(* IEC 61131-3 sources: elnaProjects/ElpcLogic/PomarKc7Changed/build_USO_ecl (part 5) *)

  (* Отключение МВ1 от КНА   *)
  stSs_Ini(data_Ini := true, inverse:=TRUE, (*wait_time:=T#0S,*) str_SS := IM.SingleSignals.Nalichie_BP5);
  inits := inits + BOOL_TO_UINT(stSs_Ini.Init);

  (* Отключение МВ1 от КНА   *)
  stSs_Ini(data_Ini := true, inverse:=TRUE, (*wait_time:=T#0S,*) str_SS := IM.SingleSignals.Nalichie_BP6);
  inits := inits + BOOL_TO_UINT(stSs_Ini.Init);

  (* Отключение МВ1 от КНА   *)
  stSs_Ini(data_Ini := true, inverse:=TRUE, (*wait_time:=T#0S,*) str_SS := IM.SingleSignals.Nalichie_BP7_BP8);
  inits := inits + BOOL_TO_UINT(stSs_Ini.Init);

  (* Отключение МВ1 от КНА   *)
  stSs_Ini(data_Ini := true, inverse:=TRUE, (*wait_time:=T#0S,*) str_SS := IM.SingleSignals.Nalichie_BP9_BP10);
  inits := inits + BOOL_TO_UINT(stSs_Ini.Init);

  (* Отключение МВ1 от КНА   *)
  stSs_Ini(data_Ini := true, inverse:=TRUE, (*wait_time:=T#0S,*) str_SS := IM.SingleSignals.Nalichie_cepei_upravlen_mv);
  inits := inits + BOOL_TO_UINT(stSs_Ini.Init);

  (* Отключение МВ1 от КНА   *)
  stSs_Ini(data_Ini := true, inverse:=TRUE, (*wait_time:=T#0S,*) str_SS := IM.SingleSignals.Nalichie_220BEAO);
  inits := inits + BOOL_TO_UINT(stSs_Ini.Init);

  (* Отключение МВ1 от КНА   *)
  stSs_Ini(data_Ini := true, inverse:=TRUE, (*wait_time:=T#0S,*) str_SS := IM.SingleSignals.Nalichie_per_220_na_vhode);
  inits := inits + BOOL_TO_UINT(stSs_Ini.Init);

  (* Отключение МВ1 от КНА   *)
  stSs_Ini(data_Ini := true, inverse:=TRUE, (*wait_time:=T#0S,*) str_SS := IM.SingleSignals.Nalichie_post_220_na_vhode);
  inits := inits + BOOL_TO_UINT(stSs_Ini.Init);

  (* Отключение МВ1 от КНА   *)
  stSs_Ini(data_Ini := true, inverse:=TRUE, (*wait_time:=T#0S,*) str_SS := IM.SingleSignals.Nalichie_BP11);
  inits := inits + BOOL_TO_UINT(stSs_Ini.Init);

  (* Отключение МВ1 от КНА   *)
  stSs_Ini(data_Ini := true, inverse:=TRUE, (*wait_time:=T#0S,*) str_SS := IM.SingleSignals.Nalichie_BP12);
  inits := inits + BOOL_TO_UINT(stSs_Ini.Init);

  (* Отключение МВ1 от КНА   *)
  stSs_Ini(data_Ini := true, inverse:=TRUE, (*wait_time:=T#0S,*) str_SS := IM.SingleSignals.Dver_SHU_pered_otkrita);
  inits := inits + BOOL_TO_UINT(stSs_Ini.Init);

  (* Отключение МВ1 от КНА   *)
  stSs_Ini(data_Ini := true, inverse:=TRUE, (*wait_time:=T#0S,*) str_SS := IM.SingleSignals.Dver_SHU_zad_otkrita);
  inits := inits + BOOL_TO_UINT(stSs_Ini.Init);

  (* Отключение МВ1 от КНА   *)
  stSs_Ini(data_Ini := true, inverse:=TRUE, (*wait_time:=T#0S,*) str_SS := IM.SingleSignals.EO_GPA_ot_knopki_SHU);
  inits := inits + BOOL_TO_UINT(stSs_Ini.Init);

  (* Отключение МВ1 от КНА   *)
  stSs_Ini(data_Ini := true, inverse:=TRUE, (*wait_time:=T#0S,*) str_SS := IM.SingleSignals.EO_EGPA_ot_PRY);
  inits := inits + BOOL_TO_UINT(stSs_Ini.Init);

  (* Отключение МВ1 от КНА   *)
  stSs_Ini(data_Ini := true, inverse:=TRUE, (*wait_time:=T#0S,*) str_SS := IM.SingleSignals.Synchroniz_rezhima_K1);
  inits := inits + BOOL_TO_UINT(stSs_Ini.Init);

                                       (* Стартовая инициализация singleOutput *)
  (* Идикация НО (подсветка кнопки на шкафу)   *)
  stSo_Ini(data_Ini := true, inOpcCommandsDisabled:=TRUE, (*wait_time:=T#0S,*) str_SO := IM.SingleOutputs.Rabota_EGPA);
  inits := inits + BOOL_TO_UINT(stSo_Ini.Init);

  (* Взвод включения БЭАО по неисправности ПТС   *)
  stSo_Ini(data_Ini := true, inOpcCommandsDisabled:=TRUE, wait_time:=T#0S, str_SO := IM.SingleOutputs.Neispr_EGPA);
  inits := inits + BOOL_TO_UINT(stSo_Ini.Init);

  (* Авария ЭГПА в КЦ   *)
  stSo_Ini(data_Ini := true, inOpcCommandsDisabled:=TRUE, (*wait_time:=T#0S,*) str_SO := IM.SingleOutputs.Avary_EGPA);
  inits := inits + BOOL_TO_UINT(stSo_Ini.Init);

  (* Авария ЭГПА в КЦ   *)
  stSo_Ini(data_Ini := true, inOpcCommandsDisabled:=TRUE, (*wait_time:=T#0S,*) str_SO := IM.SingleOutputs.U_lamp_SHU);
  inits := inits + BOOL_TO_UINT(stSo_Ini.Init);

  (* Индикация ПС Фонарь   *)
  stSo_Ini(data_Ini := true, inOpcCommandsDisabled:=TRUE, (*wait_time:=T#0S,*) str_SO := IM.SingleOutputs.AO_knopka_ind);
  inits := inits + BOOL_TO_UINT(stSo_Ini.Init);

  (* Индикация АС Фонарь   *)
  stSo_Ini(data_Ini := true, inOpcCommandsDisabled:=TRUE, (*wait_time:=T#0S,*) str_SO := IM.SingleOutputs.Pusk_SHUP);
  inits := inits + BOOL_TO_UINT(stSo_Ini.Init);

  (* Отключение МВ1 от КНА   *)
  stSo_Ini(data_Ini := true, inOpcCommandsDisabled:=TRUE, (*wait_time:=T#0S,*) str_SO := IM.SingleOutputs.Stop_SHUP);
  inits := inits + BOOL_TO_UINT(stSo_Ini.Init);

  (* Отключение МВ1 от КНА   *)
  stSo_Ini(data_Ini := true, inOpcCommandsDisabled:=TRUE, (*wait_time:=T#0S,*) str_SO := IM.SingleOutputs.NO_fonar);
  inits := inits + BOOL_TO_UINT(stSo_Ini.Init);

  (* Отключение МВ1 от КНА   *)
  stSo_Ini(data_Ini := true, inOpcCommandsDisabled:=TRUE, (*wait_time:=T#0S,*) str_SO := IM.SingleOutputs.PC_fonar);
  inits := inits + BOOL_TO_UINT(stSo_Ini.Init);

  (* Отключение МВ1 от КНА   *)
  stSo_Ini(data_Ini := true, inOpcCommandsDisabled:=TRUE, (*wait_time:=T#0S,*) str_SO := IM.SingleOutputs.AC_fonar);
  inits := inits + BOOL_TO_UINT(stSo_Ini.Init);

  (* Отключение МВ1 от КНА   *)
  stSo_Ini(data_Ini := true, inOpcCommandsDisabled:=TRUE, (*wait_time:=T#0S,*) str_SO := IM.SingleOutputs.Kr1_smazka);
  inits := inits + BOOL_TO_UINT(stSo_Ini.Init);

  (* Отключение МВ1 от КНА   *)
  stSo_Ini(data_Ini := true, inOpcCommandsDisabled:=TRUE, (*wait_time:=T#0S,*) str_SO := IM.SingleOutputs.Kr2_smazka);
  inits := inits + BOOL_TO_UINT(stSo_Ini.Init);

  (* Отключение МВ1 от КНА   *)
  stSo_Ini(data_Ini := true, inOpcCommandsDisabled:=TRUE, (*wait_time:=T#0S,*) str_SO := IM.SingleOutputs.Kr4_open_from_alg);
  inits := inits + BOOL_TO_UINT(stSo_Ini.Init);

  (* Отключение МВ1 от КНА   *)
  stSo_Ini(data_Ini := true, inOpcCommandsDisabled:=TRUE, (*wait_time:=T#0S,*) str_SO := IM.SingleOutputs.Synch_rej_K1);
  inits := inits + BOOL_TO_UINT(stSo_Ini.Init);
  initiales := 0;

  IF init THEN initiales := inits; END_IF;
END_FUNCTION_BLOCK

FUNCTION resetAndDisable : BOOL
  VAR_IN_OUT
    alg : struct_Alg;
  END_VAR
  VAR CONSTANT
    cmdReset : WORD          := 2;
  END_VAR

  IF alg.isRuning THEN
                      alg.inOpcCommandsDisabled:=TRUE;
  		alg.inCommand_Alg:=cmdReset;
  END_IF;

   alg.inCanRun:=FALSE;
END_FUNCTION

FUNCTION_BLOCK fb_puskOilSystemAlg
  VAR_IN_OUT
    StrAlg : struct_Alg;
  END_VAR
  VAR
    pnsOn : struct_PhaseAlgoritm;
    LowOil : struct_PhaseAlgoritm;
    BreakPuskTimer_Poil : struct_PhaseAlgoritm;
    Poil_DefenseActive : struct_PhaseAlgoritm;
    autoNuOn : struct_PhaseAlgoritm;
    nuOn : struct_PhaseAlgoritm;
    nu1On : struct_PhaseAlgoritm;
    nu2On : struct_PhaseAlgoritm;
    di_dPmg : struct_PhaseAlgoritm;
    dP_oilGas100 : struct_PhaseAlgoritm;
    runProtect_dP : struct_PhaseAlgoritm;
    testUnsuccessful : struct_PhaseAlgoritm;
    fb_pnsOn : fb_ph_Switch;
    fb_LowOil : fb_ph_WaitAnalogValue;
    fb_BreakPuskTimer_Poil : fb_ph_Timer;
    fb_Poil_DefenseActive : fb_ph_CustomPhase;
    fb_nuOn : fb_ph_CustomPhase;
    fb_nu1On : fb_ph_OilPump;
    fb_nu2On : fb_ph_OilPump;
    fb_autoNuOn : fb_ph_algoritm;
    fb_di_dPmg : fb_ph_CustomPhase;
    fb_dP_oilGas100 : fb_ph_WaitAnalogValue;
    fb_runProtect_dP : fb_ph_CustomPhase;
    fb_testUnsuccessful : fb_ph_CustomPhase;
    _sunpackerCommand : fb_sunpackerCommand;
    _statusAi : TYPE_StatusAi;
    _Answers : TYPE_Answers;
    _statusDualInput : TYPE_statusDualInput;
    _DualStateImAction : TYPE_DualStateImAction;
    _PhaseAlgoritmAction : TYPE_PhaseAlgoritmAction;
    source : BYTE;
    cmd : BYTE;
    lastCmd : BYTE;
    source_for_Status : BYTE;
    cmd_for_Status : BYTE;
    command_error_for_Status : BYTE;
    resetCmdTimer : TON;
    resetCmdTimerPriznak : BOOL;
    onInit : BOOL;
    waitReset : TON;
  END_VAR
  VAR_EXTERNAL
    IM : ImConfig;
    algoritms : AlgoritmsConfig;
    ai : AiConfig;
    protections : ProtectionsConfig;
    AlgTimers : struct_AlgTimers;
  END_VAR

  IF NOT onInit THEN
                 fb_pnsOn(phaseNumber:=0, act:=_on);
                fb_LowOil(phaseNumber:=1);
   fb_BreakPuskTimer_Poil(phaseNumber:=3, delay:=T#240S);
    fb_Poil_DefenseActive(phaseNumber:=5);
                  fb_nuOn(phaseNumber:=6);
                 fb_nu1On(phaseNumber:=11, act:=_on);
                 fb_nu2On(phaseNumber:=12, act:=_on);
              fb_autoNuOn(phaseNumber:=7, act:=_run, waitCompletion:=FALSE);
               fb_di_dPmg(phaseNumber:=8);
          fb_dP_oilGas100(phaseNumber:=9);
         fb_runProtect_dP(phaseNumber:=10);
      fb_testUnsuccessful(phaseNumber:=17);

  onInit:=TRUE;
  END_IF;

                fb_pnsOn(StrPh:=pnsOn, Im:=IM.pns);
               (*fb_LowOil(StrPh:=LowOil, ai:=ai.Pmasla_posle_GNS, more:=im.AutoPns_UstRun.Value);*)
  fb_BreakPuskTimer_Poil(StrPh:=BreakPuskTimer_Poil, timer:=AlgTimers.puskOilSystem_BreakPuskTimer_Poil);
   fb_Poil_DefenseActive(StrPh:=Poil_DefenseActive);
                 fb_nuOn(StrPh:=nuOn);
                fb_nu1On(StrPh:=nu1On, Im:=Im.nu1);
                fb_nu2On(StrPh:=nu2On, Im:=Im.nu2);
             fb_autoNuOn(StrPh:=autoNuOn, alg:=algoritms.autoNu);
              fb_di_dPmg(StrPh:=di_dPmg);
         (*fb_dP_oilGas100(StrPh:=dP_oilGas100, ai:=ai.Tmasla_MB, more:=im.PuskOilSystem_UstdPmg.Value);*)
        fb_runProtect_dP(StrPh:=runProtect_dP);
     fb_testUnsuccessful(StrPh:=testUnsuccessful);

  IF StrAlg.isRuning THEN

      StrAlg.hasError := LowOil.error OR dP_oilGas100.error OR pnsOn.error OR testUnsuccessful.error;

      IF pnsOn.top THEN
          runPhase(LowOil);
      END_IF;

      IF LowOil.top THEN
          runAiProtection(protections.Os_sdvig_nagnetatelja_minus);
          (*runDiProtection(protections.Vibro_skorost_OP_shesterni_RED_T6);*)
          runPhase(Poil_DefenseActive);
          (*IM.SingleSignals.P_oil_low.Disabled_Sig:=FALSE;*)
          ai.Pmasla_posle_GNS.Disabled_LA:=FALSE;
          ai.Pmasla_posle_GNS.Disabled_LW:=FALSE;
          ai.Pmasla_posle_NU.Disabled_LW:=FALSE;
      END_IF;

      IF Poil_DefenseActive.start AND NOT Poil_DefenseActive.top THEN
         Poil_DefenseActive.top:=protections.Os_sdvig_nagnetatelja_minus.isRunning AND protections.Vibro_skorost_OP_shesterni_RED_T6.isRunning;
      END_IF;

      IF Poil_DefenseActive.top THEN
         (* runPhase(autoNuOn);*)
  	runPhase(nuOn);
      END_IF;

      IF nuOn.start AND NOT nuOn.top THEN
         (* IF IM.SingleOutputs.Value = 0 THEN
              runPhase(nu1On);
          END_IF;

          IF IM.SingleOutputs.Value = 1 THEN
              runPhase(nu2On);
          END_IF;*)
         nuOn.top:= Im.nu1.onStatus = _statusDualInput.STATUS_ON OR Im.nu2.onStatus = _statusDualInput.STATUS_ON;
      END_IF;

      IF nuOn.top THEN
  	runPhase(di_dPmg);
            runPhase(dP_oilGas100);
      END_IF;

      (*IF di_dPmg.start AND NOT di_dPmg.top THEN
         di_dPmg.top:= NOT IM.SingleSignals.dP_oilgaz_low.Q;
      END_IF;*)

      IF dP_oilGas100.top AND di_dPmg.top THEN
            runPhase(autoNuOn);
  	runPhase(runProtect_dP);
  	runAiProtection(protections.Os_sdvig_nagnetatelja_plus);
            (*runDiProtection(protections.Vibro_skorost_OP_shesterni_RED_T5);
            IM.SingleSignals.dP_oilgaz_low.Disabled_Sig:=FALSE;
            ai.Tmasla_MB.Disabled_LA:=FALSE;
            ai.Tmasla_MB.Disabled_LW:=FALSE;*)
      END_IF;

      IF runProtect_dP.start AND NOT runProtect_dP.top THEN
         runProtect_dP.top:= protections.Os_sdvig_nagnetatelja_plus.isRunning AND protections.Vibro_skorost_OP_shesterni_RED_T5.isRunning;
      END_IF;

      IF BreakPuskTimer_Poil.top AND (NOT runProtect_dP.top) THEN
  	testUnsuccessful.error:=TRUE;
      END_IF;

      IF runProtect_dP.top THEN
            resetPhase(BreakPuskTimer_Poil);
  	waitReset(IN:=TRUE);
      END_IF;

      IF waitReset.Q AND NOT (algoritms.Apusk.isRuning OR algoritms.SemiAutoPusk.isRuning) THEN
      resetAndDisable(StrAlg);
      END_IF;

      StrAlg.isEnded:=runProtect_dP.top;
  END_IF;

  StrAlg.CanRun := StrAlg.inCanRun;
  StrAlg.OpcCommandsDisabled := StrAlg.inOpcCommandsDisabled;

  (* ---- Если управление с ВУ заблокировано, то  передаем команду из алгоритма ---- *)
  IF StrAlg.inOpcCommandsDisabled THEN
  	StrAlg.inCommand := StrAlg.inCommand_Alg;
  ELSE (* иначе передаем команду с АРМа*)
  	StrAlg.inCommand := StrAlg.inCommand_ARM;
  END_IF;

  _sunpackerCommand(command := StrAlg.inCommand);
  	source := _sunpackerCommand.source;
  	cmd := _sunpackerCommand.cmd;

  IF cmd <> 0 AND lastCmd <> cmd AND (((NOT StrAlg.opcCommandsDisabled) AND source > 0) OR source = 0) then
  	CASE BYTE_TO_INT(cmd) OF
  		(*cmdRun*) 1: 	IF (StrAlg.CanRun) THEN
  					StrAlg.isRuning := TRUE;
  					StrAlg.isEnded := FALSE;
  					StrAlg.hasError := FALSE;
  					(*****************       OnRun       *****************)
                                                    runPhase(pnsOn);
                                                    runPhase(BreakPuskTimer_Poil);
                                                    runPhase(testUnsuccessful);
  					cmd_for_Status := cmd;
  					source_for_Status := source;
  					command_error_for_Status := 0;
  				ELSE
  					StrAlg.isRuning := FALSE;
  					StrAlg.isEnded := FALSE;
  					StrAlg.hasError 	:= FALSE;

  					cmd_for_Status := 0;
  					source_for_Status := source;
  					command_error_for_Status := cmd;
  				END_IF;
  		(*cmdReset*) 2: 	StrAlg.isRuning := FALSE;
  				StrAlg.isEnded := FALSE;
  				StrAlg.hasError 	:= FALSE;

                                           (*****************       OnReset       *****************)
                                          waitReset(IN:=FALSE);
                                          resetPhase(pnsOn);
                                          resetPhase(LowOil);
                                          resetPhase(BreakPuskTimer_Poil);
                                          resetPhase(Poil_DefenseActive);
                                          resetPhase(autoNuOn);
                                          resetPhase(nu1On);
                                          resetPhase(nu2On);
                                          resetPhase(nuOn);
                                          resetPhase(di_dPmg);
                                          resetPhase(dP_oilGas100);
                                          resetPhase(runProtect_dP);
                                          resetPhase(testUnsuccessful);
  	                              (*protections.Os_sdvig_nagnetatelja_minus.inOpcCommandsDisabled:=FALSE;
                                          protections.Vibro_skorost_OP_shesterni_RED_T6.inOpcCommandsDisabled:=FALSE;
                                          protections.Os_sdvig_nagnetatelja_plus.inOpcCommandsDisabled:=FALSE;
                                          protections.Vibro_skorost_OP_shesterni_RED_T5.inOpcCommandsDisabled:=FALSE;*)

  				cmd_for_Status := cmd;
  				source_for_Status := source;
  				command_error_for_Status := 0;
  	END_CASE;
  	resetCmdTimer(IN := false);
  	resetCmdTimerPriznak := TRUE;
  END_IF;
  lastCmd := cmd;

  resetCmdTimer(IN := resetCmdTimerPriznak, PT := T#5S);
  IF resetCmdTimer.Q THEN
  	resetCmdTimerPriznak := FALSE;
  	source_for_Status := 0;
  	cmd_for_Status := 0;
  	command_error_for_Status := 0;
  END_IF;

  StrAlg.Start:= pnsOn.startStatus
              OR LowOil.startStatus
              OR BreakPuskTimer_Poil.startStatus
              OR Poil_DefenseActive.startStatus
              OR nuOn.startStatus
              OR di_dPmg.startStatus
              OR dP_oilGas100.startStatus
              OR runProtect_dP.startStatus
              OR testUnsuccessful.startStatus;

  StrAlg.Error:= pnsOn.errorStatus
              OR LowOil.errorStatus
              OR BreakPuskTimer_Poil.errorStatus
              OR Poil_DefenseActive.errorStatus
              OR nuOn.errorStatus
              OR di_dPmg.errorStatus
              OR dP_oilGas100.errorStatus
              OR runProtect_dP.errorStatus
              OR testUnsuccessful.errorStatus;

  StrAlg.Top:=   pnsOn.topStatus
              OR LowOil.topStatus
              OR BreakPuskTimer_Poil.topStatus
              OR Poil_DefenseActive.topStatus
              OR nuOn.topStatus
              OR di_dPmg.topStatus
              OR dP_oilGas100.topStatus
              OR runProtect_dP.topStatus
              OR testUnsuccessful.topStatus;

  (*TODO: TYPE PROGRAM CODE HERE*)
  StrAlg.status :=  SHL(BYTE_TO_DWORD(source_for_Status), 29)
  			OR SHL(BYTE_TO_DWORD(cmd_for_Status), 26)
  			OR SHL(BYTE_TO_DWORD(command_error_for_Status), 23)
  			OR SHL(BOOL_TO_DWORD(StrAlg.OpcCommandsDisabled ), 21)
  			OR SHL(BOOL_TO_DWORD(StrAlg.hasError),4)
  			OR SHL(BOOL_TO_DWORD(StrAlg.CanRun),2)
  			OR SHL(BOOL_TO_DWORD(StrAlg.isEnded),1)
  			OR BOOL_TO_DWORD(StrAlg.isRuning);
END_FUNCTION_BLOCK

FUNCTION BlockAllIM : BOOL
  VAR_IN_OUT
    IM : ImConfig;
  END_VAR

  IF NOT IM.Kran1.inOpcCommandsDisabled   THEN IM.Kran1.inOpcCommandsDisabled:=TRUE; END_IF;
  IF NOT IM.Kran2.inOpcCommandsDisabled   THEN IM.Kran2.inOpcCommandsDisabled:=TRUE; END_IF;
  IF NOT IM.Kran3b.inOpcCommandsDisabled  THEN IM.Kran3b.inOpcCommandsDisabled:=TRUE; END_IF;
  IF NOT IM.Kran4.inOpcCommandsDisabled   THEN IM.Kran4.inOpcCommandsDisabled:=TRUE; END_IF;
  IF NOT IM.Kran5.inOpcCommandsDisabled   THEN IM.Kran5.inOpcCommandsDisabled:=TRUE; END_IF;
  (*IF NOT IM.Kran6.inOpcCommandsDisabled   THEN IM.Kran6.inOpcCommandsDisabled:=TRUE; END_IF;*)

  IF NOT IM.nu1.inOpcCommandsDisabled     THEN IM.nu1.inOpcCommandsDisabled:=TRUE; END_IF;
  IF NOT IM.nu2.inOpcCommandsDisabled     THEN IM.nu2.inOpcCommandsDisabled:=TRUE; END_IF;
  IF NOT IM.pns.inOpcCommandsDisabled     THEN IM.pns.inOpcCommandsDisabled:=TRUE; END_IF;
  IF NOT IM.v1_Avom.inOpcCommandsDisabled THEN IM.v1_Avom.inOpcCommandsDisabled:=TRUE; END_IF;
  IF NOT IM.v2_Avom.inOpcCommandsDisabled THEN IM.v2_Avom.inOpcCommandsDisabled:=TRUE; END_IF;
  (*IF NOT IM.Ten.inOpcCommandsDisabled     THEN IM.Ten.inOpcCommandsDisabled:=TRUE; END_IF;*)
  IF NOT IM.mv.inOpcCommandsDisabled      THEN IM.mv.inOpcCommandsDisabled:=TRUE; END_IF;
END_FUNCTION

FUNCTION UnBlockAllIM : BOOL
  VAR_IN_OUT
    IM : ImConfig;
  END_VAR

  (*IF IM.TypeSwitch.Value = 1 THEN*)

  IF IM.Kran1.inOpcCommandsDisabled   THEN IM.Kran1.inOpcCommandsDisabled:=FALSE; END_IF;
  IF IM.Kran2.inOpcCommandsDisabled   THEN IM.Kran2.inOpcCommandsDisabled:=FALSE; END_IF;
  IF IM.Kran3b.inOpcCommandsDisabled  THEN IM.Kran3b.inOpcCommandsDisabled:=FALSE; END_IF;
  IF IM.Kran4.inOpcCommandsDisabled   THEN IM.Kran4.inOpcCommandsDisabled:=FALSE; END_IF;
  IF IM.Kran5.inOpcCommandsDisabled   THEN IM.Kran5.inOpcCommandsDisabled:=FALSE; END_IF;
  (*IF IM.Kran6.inOpcCommandsDisabled   THEN IM.Kran6.inOpcCommandsDisabled:=FALSE; END_IF;*)
  (*END_IF;*)

  IF IM.nu1.inOpcCommandsDisabled     THEN IM.nu1.inOpcCommandsDisabled:=FALSE; END_IF;
  IF IM.nu2.inOpcCommandsDisabled     THEN IM.nu2.inOpcCommandsDisabled:=FALSE; END_IF;
  IF IM.pns.inOpcCommandsDisabled     THEN IM.pns.inOpcCommandsDisabled:=FALSE; END_IF;
  IF IM.v1_Avom.inOpcCommandsDisabled THEN IM.v1_Avom.inOpcCommandsDisabled:=FALSE; END_IF;
  IF IM.v2_Avom.inOpcCommandsDisabled THEN IM.v2_Avom.inOpcCommandsDisabled:=FALSE; END_IF;
  (*IF IM.Ten.inOpcCommandsDisabled     THEN IM.Ten.inOpcCommandsDisabled:=FALSE; END_IF;*)
  IF IM.mv.inOpcCommandsDisabled      THEN IM.mv.inOpcCommandsDisabled:=FALSE; END_IF;
END_FUNCTION

FUNCTION_BLOCK TestImAlg
  VAR_IN_OUT
    StrAlg : struct_Alg;
  END_VAR
  VAR
    _sunpackerCommand : fb_sunpackerCommand;
    source : BYTE;
    cmd : BYTE;
    lastCmd : BYTE;
    source_for_Status : BYTE;
    cmd_for_Status : BYTE;
    command_error_for_Status : BYTE;
    resetCmdTimer : TON;
    resetCmdTimerPriznak : BOOL;
  END_VAR
  VAR_EXTERNAL
    protectManager : struct_ProtectionsManager;
    algManager : struct_AlgoritmsManager;
    ModeGpa : TYPE_ModeGpa;
    PMcommand : TYPE_CommandsPotectionsManager;
    IM : ImConfig;
  END_VAR

  StrAlg.CanRun := StrAlg.inCanRun;
  StrAlg.OpcCommandsDisabled := StrAlg.inOpcCommandsDisabled;

  (* ---- Если управление с ВУ заблокировано, то передаем команду из алгоритма ---- *)
  IF StrAlg.inOpcCommandsDisabled THEN
  	StrAlg.inCommand := StrAlg.inCommand_Alg;
  ELSE (* иначе передаем команду с АРМа*)
  	StrAlg.inCommand := StrAlg.inCommand_ARM;
  END_IF;

  _sunpackerCommand(command := StrAlg.inCommand);
  	source := _sunpackerCommand.source;
  	cmd := _sunpackerCommand.cmd;

  IF cmd <> 0 AND lastCmd <> cmd AND (((NOT StrAlg.opcCommandsDisabled) AND source > 0) OR source = 0) then
  	CASE BYTE_TO_INT(cmd) OF
  		(*cmdRun*) 1: 	IF (StrAlg.CanRun) THEN
  					StrAlg.isRuning := TRUE;
  					StrAlg.isEnded := FALSE;
  					StrAlg.hasError 	:= FALSE;
                                               (*****************       OnRun       *****************)

                                                        algManager.nMode:=ModeGpa.MODE_TESTIM;
  					    UnBlockAllIM(IM);

                                                    (*StrAlg.inOpcCommandsDisabled:=FALSE;*)
  					cmd_for_Status := cmd;
  					source_for_Status := source;
  					command_error_for_Status := 0;
  				ELSE
  					StrAlg.isRuning := FALSE;
  					StrAlg.isEnded := FALSE;
  					StrAlg.hasError 	:= FALSE;

  					cmd_for_Status := 0;
  					source_for_Status := source;
  					command_error_for_Status := cmd;
  				END_IF;
  		(*cmdReset*) 2: 	StrAlg.isRuning := FALSE;
  				StrAlg.isEnded := FALSE;
  				StrAlg.hasError 	:= FALSE;
                                          (*****************       OnReset       *****************)
                                                    BlockAllIM(IM);
                                                    algManager.nMode:=ModeGpa.MODE_STOP;

  				cmd_for_Status := cmd;
  				source_for_Status := source;
  				command_error_for_Status := 0;
  	END_CASE;
  	resetCmdTimer(IN := false);
  	resetCmdTimerPriznak := TRUE;
  END_IF;
  lastCmd := cmd;

  resetCmdTimer(IN := resetCmdTimerPriznak, PT := T#5S);
  IF resetCmdTimer.Q THEN
  	resetCmdTimerPriznak := FALSE;
  	source_for_Status := 0;
  	cmd_for_Status := 0;
  	command_error_for_Status := 0;
  END_IF;

  StrAlg.status :=  SHL(BYTE_TO_DWORD(source_for_Status), 29)
  			OR SHL(BYTE_TO_DWORD(cmd_for_Status), 26)
  			OR SHL(BYTE_TO_DWORD(command_error_for_Status), 23)
  			OR SHL(BOOL_TO_DWORD(StrAlg.OpcCommandsDisabled ), 21)
  			OR SHL(BOOL_TO_DWORD(StrAlg.hasError),4)
  			OR SHL(BOOL_TO_DWORD(StrAlg.CanRun),2)
  			OR SHL(BOOL_TO_DWORD(StrAlg.isEnded),1)
  			OR BOOL_TO_DWORD(StrAlg.isRuning);
END_FUNCTION_BLOCK

FUNCTION askQuestion : BOOL
  VAR_IN_OUT
    StrQ : struct_Question;
  END_VAR

  IF NOT StrQ.ask THEN
                      StrQ.inOpcCommandsDisabled:=FALSE;
                      StrQ.ask:=TRUE;
  END_IF;
END_FUNCTION

FUNCTION resetQuestion : BOOL
  VAR_IN_OUT
    StrQ : struct_Question;
  END_VAR

  IF StrQ.ask THEN
                      StrQ.inOpcCommandsDisabled:=TRUE;
                      StrQ.reset:=TRUE;
  END_IF;
END_FUNCTION

FUNCTION_BLOCK testdPmgAlg
  VAR_IN_OUT
    StrAlg : struct_Alg;
  END_VAR
  VAR
    puskOilSystem : struct_PhaseAlgoritm;
  END_VAR
  VAR_IN_OUT
    algContinue : struct_Question;
  END_VAR
  VAR
    nuOff : struct_PhaseAlgoritm;
    dPmgAi : struct_PhaseAlgoritm;
    dPmgDi : struct_PhaseAlgoritm;
    nuOn : struct_PhaseAlgoritm;
    noRezrv : struct_PhaseAlgoritm;
    BreakTest : struct_PhaseAlgoritm;
    testUnsuccessful : struct_PhaseAlgoritm;
    pnsOff : struct_PhaseAlgoritm;
    stopANU : struct_PhaseAlgoritm;
    Ust_dPLow : struct_PhaseAlgoritm;
    nu1Off : struct_PhaseAlgoritm;
    nu2Off : struct_PhaseAlgoritm;
    stopNU1 : struct_PhaseAlgoritm;
    stopNU2 : struct_PhaseAlgoritm;
    fb_puskOilSystem : fb_ph_algoritm;
    fb_algContinue : fb_Question;
    fb_nuOff : fb_ph_CustomPhase;
    fb_dPmgAi : fb_ph_WaitAnalogValue;
    fb_dPmgDi : fb_ph_CustomPhase;
    fb_nuOn : fb_ph_CustomPhase;
    fb_noRezrv : fb_ph_CustomPhase;
    fb_BreakTest : fb_ph_Timer;
    fb_testUnsuccessful : fb_ph_CustomPhase;
    fb_pnsOff : fb_ph_Switch;
    fb_stopANU : fb_ph_CustomPhase;
    fb_nu1Off : fb_ph_OilPump;
    fb_nu2Off : fb_ph_OilPump;
    fb_stopNU1 : fb_ph_OilPump;
    fb_stopNU2 : fb_ph_OilPump;
    _sunpackerCommand : fb_sunpackerCommand;
    _DualStateImAction : TYPE_DualStateImAction;
    _Answers : TYPE_Answers;
    _statusDualInput : TYPE_statusDualInput;
    _StatusAi : TYPE_StatusAi;
    _PhaseAlgoritmAction : TYPE_PhaseAlgoritmAction;
    source : BYTE;
    cmd : BYTE;
    lastCmd : BYTE;
    source_for_Status : BYTE;
    cmd_for_Status : BYTE;
    command_error_for_Status : BYTE;
    resetCmdTimer : TON;
    resetCmdTimerPriznak : BOOL;
    onInit : BOOL;
    _resetQuestion : BOOL;
    waitReset : TON;
    WaitOnNU : TON;
  END_VAR
  VAR_EXTERNAL
    IM : ImConfig;
    algoritms : AlgoritmsConfig;
    ai : AiConfig;
    AlgTimers : struct_AlgTimers;
    ModeGpa : TYPE_ModeGpa;
    algManager : struct_AlgoritmsManager;
    protections : ProtectionsConfig;
    NotHasRezervNU : BOOL;
  END_VAR

  IF NOT onInit THEN

      fb_puskOilSystem(phaseNumber:=0, act:=_run, waitCompletion:=TRUE);
          algContinue.AnswerVariants:=_Answers.ANS_YES;
              fb_nuOff(phaseNumber:=1);
             fb_dPmgAi(phaseNumber:=2);
             fb_dPmgDi(phaseNumber:=3);
               fb_nuOn(phaseNumber:=4);
            fb_noRezrv(phaseNumber:=5);
   fb_testUnsuccessful(phaseNumber:=6);
          fb_BreakTest(phaseNumber:=7, delay:=T#10S);
             fb_pnsOff(phaseNumber:=8, act:=_off);
            fb_stopANU(phaseNumber:=9);
             fb_nu1Off(phaseNumber:=11, act:=_off);
             fb_nu2Off(phaseNumber:=12, act:=_off);
            fb_stopNU1(phaseNumber:=15, act:=_off);
            fb_stopNU2(phaseNumber:=16, act:=_off);
  onInit:=TRUE;
  END_IF;

      fb_puskOilSystem(StrPh:=puskOilSystem, alg:=algoritms.puskOilSystem);
        fb_algContinue(StrQ:=algContinue);
              fb_nuOff(StrPh:=nuOff);
             (*fb_dPmgAi(StrPh:=dPmgAi, ai:=ai.Tmasla_MB, less:=im.testdPmg_Ust_dPLow.Value);*)
             fb_dPmgDi(StrPh:=dPmgDi);
               fb_nuOn(StrPh:=nuOn);
            fb_noRezrv(StrPh:=noRezrv);
   fb_testUnsuccessful(StrPh:=testUnsuccessful);
          fb_BreakTest(StrPh:=BreakTest, timer:=AlgTimers.testdPmg_BreakTest);
             fb_pnsOff(StrPh:=pnsOff, Im:=Im.pns);
            fb_stopANU(StrPh:=stopANU);
             fb_nu1Off(StrPh:=nu1Off, Im:=Im.nu1);
             fb_nu2Off(StrPh:=nu2Off, Im:=Im.nu2);
            fb_stopNU1(StrPh:=stopNU1, Im:=Im.nu1);
            fb_stopNU2(StrPh:=stopNU2, Im:=Im.nu2);

  StrAlg.CanRun := StrAlg.inCanRun;
  StrAlg.OpcCommandsDisabled := StrAlg.inOpcCommandsDisabled;

  IF StrAlg.isRuning THEN

      StrAlg.hasError := pnsOff.error OR nu1Off.error OR nu2Off.error
      OR stopNU1.error OR stopNU2.error OR testUnsuccessful.error;

      IF puskOilSystem.top THEN
           IF NOT _resetQuestion THEN
           askQuestion(algContinue);
            _resetQuestion:=TRUE;
           END_IF;
      END_IF;

      IF algContinue.answer = _Answers.ANS_YES AND NOT nuOff.top THEN

          runPhase(nuOff);

          IF Im.nu1.onStatus = _statusDualInput.STATUS_ON THEN
  		runPhase(nu1Off);
          END_IF;

          IF Im.nu2.onStatus = _statusDualInput.STATUS_ON THEN
  		runPhase(nu2Off);
          END_IF;

          resetQuestion(algContinue);

      END_IF;

      IF nuOff.start AND NOT nuOff.top THEN
            runPhase(BreakTest);
  	nuOff.top:= Im.nu1.onStatus = _statusDualInput.STATUS_Off
                    AND Im.nu2.onStatus = _statusDualInput.STATUS_Off;
      END_IF;

      IF nuOff.top THEN

          runPhase(dPmgAi);
          runPhase(dPmgDi);
      END_IF;

      (*IF dPmgDi.start AND NOT dPmgDi.top THEN
          dPmgDi.top:=Im.SingleSignals.dP_oilgaz_low.q;
      END_IF;*)

      IF dPmgAi.top AND dPmgDi.top THEN
          runPhase(nuOn);
          runPhase(noRezrv);
      END_IF;

      IF noRezrv.start AND NOT noRezrv.top THEN
          noRezrv.top:=NotHasRezervNU;
      END_IF;

       IF nuOn.start AND (NOT WaitOnNU.Q) THEN
          WaitOnNU(IN:=Im.nu1.onStatus = _statusDualInput.STATUS_On OR
              Im.nu2.onStatus = _statusDualInput.STATUS_On, PT:=T#2S);
          nuOn.top:=Im.nu1.onStatus = _statusDualInput.STATUS_On OR
              Im.nu2.onStatus = _statusDualInput.STATUS_On;
      END_IF;

      IF  WaitOnNU.Q AND noRezrv.top THEN
          ai.Tmasla_MB.Disabled_LA:=TRUE;
          ai.Tmasla_MB.Disabled_LW:=TRUE;
          (*IM.SingleSignals.dP_oilgaz_low.Disabled_Sig:=TRUE;
          IM.SingleSignals.P_oil_low.Disabled_Sig:=TRUE;*)
          ai.Pmasla_posle_GNS.Disabled_LA:=TRUE;
          ai.Pmasla_posle_GNS.Disabled_LW:=TRUE;
          ai.Pmasla_posle_NU.Disabled_LW:=TRUE;

          resetAiProtection(protections.Os_sdvig_nagnetatelja_minus);
          (*resetDiProtection(protections.Vibro_skorost_OP_shesterni_RED_T6);*)
          resetAiProtection(protections.Os_sdvig_nagnetatelja_plus);
          (*resetDiProtection(protections.Vibro_skorost_OP_shesterni_RED_T5);*)

          resetIfRunning(algoritms.autoNu);
          resetIfRunning(algoritms.AutoPns);

          runPhase(stopANU);
          runPhase(pnsOff);

          runPhase(stopNU1);
          runPhase(stopNU2);

      END_IF;

      IF stopANU.start AND NOT stopANU.top THEN

  	stopANU.top:= Im.nu1.onStatus = _statusDualInput.STATUS_Off AND
                          Im.nu2.onStatus = _statusDualInput.STATUS_Off;
      END_IF;

      IF BreakTest.top AND NOT pnsOff.top THEN
  	testUnsuccessful.error:=TRUE;
      END_IF;

      IF pnsOff.top AND stopANU.top THEN
            resetPhase(BreakTest);
  	waitReset(IN:=TRUE, PT:= T#3S);
      END_IF;

      IF waitReset.Q THEN
          algManager.nMode:=ModeGpa.MODE_STOP;
          resetIfRunning(StrAlg);
      END_IF;

      StrAlg.isEnded:= pnsOff.top AND stopANU.top;

  END_IF;

  StrAlg.CanRun := StrAlg.inCanRun;
  StrAlg.OpcCommandsDisabled := StrAlg.inOpcCommandsDisabled;

  (* ---- Если управление с ВУ заблокировано, то  передаем команду из алгоритма ---- *)
  IF StrAlg.inOpcCommandsDisabled THEN
  	StrAlg.inCommand := StrAlg.inCommand_Alg;
  ELSE (* иначе передаем команду с АРМа*)
  	StrAlg.inCommand := StrAlg.inCommand_ARM;
  END_IF;

  _sunpackerCommand(command := StrAlg.inCommand);
  	source := _sunpackerCommand.source;
  	cmd := _sunpackerCommand.cmd;

  IF cmd <> 0 AND lastCmd <> cmd AND (((NOT StrAlg.opcCommandsDisabled) AND source > 0) OR source = 0) then
  	CASE BYTE_TO_INT(cmd) OF
  		(*cmdRun*) 1: 	IF (StrAlg.CanRun) THEN
  					StrAlg.isRuning := TRUE;
  					StrAlg.isEnded := FALSE;
  					StrAlg.hasError := FALSE;
  					(*****************       OnRun       *****************)

                                                    algManager.nMode:=ModeGpa.MODE_TESTDPMG;
                                                    resetAndDisable(alg:=algoritms.ppu);
                                                    algoritms.puskOilSystem.inCanRun:= TRUE;
                                                    runPhase(puskOilSystem);

  					cmd_for_Status := cmd;
  					source_for_Status := source;
  					command_error_for_Status := 0;
  				ELSE
  					StrAlg.isRuning := FALSE;
  					StrAlg.isEnded := FALSE;
  					StrAlg.hasError 	:= FALSE;

  					cmd_for_Status := 0;
  					source_for_Status := source;
  					command_error_for_Status := cmd;
  				END_IF;
  		(*cmdReset*) 2: 	StrAlg.isRuning := FALSE;
  				StrAlg.isEnded := FALSE;
  				StrAlg.hasError 	:= FALSE;

                                           (*****************       OnReset       *****************)
                                          waitReset(IN:=FALSE);
                                          WaitOnNU(IN:=FALSE);
                                          _resetQuestion:=FALSE;
                                          ai.Pmasla_posle_GNS.Disabled_LA:=TRUE;
                                          ai.Pmasla_posle_GNS.Disabled_LW:=TRUE;
                                          ai.Pmasla_posle_NU.Disabled_LW:=TRUE;
                                          (*IM.SingleSignals.P_oil_low.Disabled_Sig:=TRUE;
                                          IM.SingleSignals.dP_oilgaz_low.Disabled_Sig:=TRUE;*)
                                          ai.Tmasla_MB.Disabled_LA:=TRUE;
                                          ai.Tmasla_MB.Disabled_LW:=TRUE;
                                          resetAiProtection(protections.Os_sdvig_nagnetatelja_minus);
                                          (*resetDiProtection(protections.Vibro_skorost_OP_shesterni_RED_T6);*)
                                          resetAiProtection(protections.Os_sdvig_nagnetatelja_plus);
                                          (*resetDiProtection(protections.Vibro_skorost_OP_shesterni_RED_T5);*)

                                          resetPhase(puskOilSystem);
                                          resetPhase(nuOff);
                                          resetPhase(dPmgAi);
                                          resetPhase(dPmgDi);
                                          resetPhase(nuOn);
                                          resetPhase(noRezrv);
                                          resetPhase(BreakTest);
                                          resetPhase(testUnsuccessful);
                                          resetPhase(pnsOff);
                                          resetPhase(stopANU);
                                          resetPhase(nu1Off);
                                          resetPhase(nu2Off);
                                          resetPhase(stopNU1);
                                          resetPhase(stopNU2);

                                          resetQuestion(algContinue);

                                          StrAlg.inOpcCommandsDisabled:=FALSE;

  				cmd_for_Status := cmd;
  				source_for_Status := source;
  				command_error_for_Status := 0;
  	END_CASE;
  	resetCmdTimer(IN := false);
  	resetCmdTimerPriznak := TRUE;
  END_IF;
  lastCmd := cmd;

  resetCmdTimer(IN := resetCmdTimerPriznak, PT := T#5S);
  IF resetCmdTimer.Q THEN
  	resetCmdTimerPriznak := FALSE;
  	source_for_Status := 0;
  	cmd_for_Status := 0;
  	command_error_for_Status := 0;
  END_IF;

  StrAlg.Start:= puskOilSystem.startStatus
              OR nuOff.startStatus
              OR dPmgAi.startStatus
              OR dPmgDi.startStatus
              OR nuOn.startStatus
              OR noRezrv.startStatus
              OR BreakTest.startStatus
              OR testUnsuccessful.startStatus
              OR pnsOff.startStatus
              OR stopANU.startStatus
              OR nu1Off.startStatus
              OR nu2Off.startStatus;

  StrAlg.Error:=  puskOilSystem.errorStatus
              OR nuOff.errorStatus
              OR dPmgAi.errorStatus
              OR dPmgDi.errorStatus
              OR nuOn.errorStatus
              OR noRezrv.errorStatus
              OR BreakTest.errorStatus
              OR testUnsuccessful.errorStatus
              OR pnsOff.errorStatus
              OR stopANU.errorStatus
              OR nu1Off.errorStatus
              OR nu2Off.errorStatus;

  StrAlg.Top:=   puskOilSystem.topStatus
              OR nuOff.topStatus
              OR dPmgAi.topStatus
              OR dPmgDi.topStatus
              OR nuOn.topStatus
              OR noRezrv.topStatus
              OR BreakTest.topStatus
              OR testUnsuccessful.topStatus
              OR pnsOff.topStatus
              OR stopANU.topStatus
              OR nu1Off.topStatus
              OR nu2Off.topStatus;

  (*TODO: TYPE PROGRAM CODE HERE*)
  StrAlg.status :=  SHL(BYTE_TO_DWORD(source_for_Status), 29)
  			OR SHL(BYTE_TO_DWORD(cmd_for_Status), 26)
  			OR SHL(BYTE_TO_DWORD(command_error_for_Status), 23)
  			OR SHL(BOOL_TO_DWORD(StrAlg.OpcCommandsDisabled ), 21)
  			OR SHL(BOOL_TO_DWORD(StrAlg.hasError),4)
  			OR SHL(BOOL_TO_DWORD(StrAlg.CanRun),2)
  			OR SHL(BOOL_TO_DWORD(StrAlg.isEnded),1)
  			OR BOOL_TO_DWORD(StrAlg.isRuning);
END_FUNCTION_BLOCK

FUNCTION_BLOCK SemiAutoPuskAlg
  VAR_IN_OUT
    StrAlg : struct_Alg;
  END_VAR
  VAR
    runOilsystem : struct_PhaseAlgoritm;
    runEngine : struct_PhaseAlgoritm;
    filling : struct_PhaseAlgoritm;
  END_VAR
  VAR_IN_OUT
    cmdRun1ph : struct_Question;
    cmdRun2ph : struct_Question;
    cmdRun3ph : struct_Question;
  END_VAR
  VAR
    fb_runOilsystem : fb_ph_algoritm;
    fb_runEngine : fb_ph_algoritm;
    fb_filling : fb_ph_algoritm;
    fb_cmdRun1ph : fb_Question;
    fb_cmdRun2ph : fb_Question;
    fb_cmdRun3ph : fb_Question;
    _sunpackerCommand : fb_sunpackerCommand;
    _PhaseAlgoritmAction : TYPE_PhaseAlgoritmAction;
    _statusDualInput : TYPE_statusDualInput;
    _Answers : TYPE_Answers;
    source : BYTE;
    cmd : BYTE;
    lastCmd : BYTE;
    source_for_Status : BYTE;
    cmd_for_Status : BYTE;
    command_error_for_Status : BYTE;
    resetCmdTimer : TON;
    resetCmdTimerPriznak : BOOL;
    onInit : BOOL;
    waitReset : TON;
  END_VAR
  VAR_EXTERNAL
    algoritms : AlgoritmsConfig;
    ModeGpa : TYPE_ModeGpa;
    algManager : struct_AlgoritmsManager;
    IM : ImConfig;
  END_VAR

  IF NOT onInit THEN
                 cmdRun1ph.AnswerVariants:=_Answers.ANS_YES;
           fb_runOilsystem(phaseNumber:=0, act:=_run, waitCompletion:=TRUE);
                 cmdRun2ph.AnswerVariants:=_Answers.ANS_YES;
              fb_runEngine(phaseNumber:=1, act:=_run, waitCompletion:=TRUE);
                 cmdRun3ph.AnswerVariants:=_Answers.ANS_YES;
                fb_filling(phaseNumber:=2, act:=_run, waitCompletion:=TRUE);

  onInit:=TRUE;
  END_IF;
              fb_cmdRun1ph(StrQ:=cmdRun1ph);
           fb_runOilsystem(StrPh:=runOilsystem, alg:=algoritms.puskOilSystem);
              fb_cmdRun2ph(StrQ:=cmdRun2ph);
              fb_runEngine(StrPh:=runEngine, alg:=algoritms.engineRun);
              fb_cmdRun3ph(StrQ:=cmdRun3ph);
                fb_filling(StrPh:=filling, alg:=algoritms.filling);

  StrAlg.CanRun := StrAlg.inCanRun;
  StrAlg.OpcCommandsDisabled := StrAlg.inOpcCommandsDisabled;

  IF StrAlg.isRuning THEN

      StrAlg.hasError := runOilsystem.error OR runEngine.error OR filling.error;

      IF cmdRun1ph.answer = _Answers.ANS_YES THEN
  	runPhase(runOilsystem);
            resetQuestion(cmdRun1ph);
      END_IF;

      IF runOilsystem.top AND NOT runEngine.start THEN
           askQuestion(cmdRun2ph);
      END_IF;

      IF cmdRun2ph.answer = _Answers.ANS_YES THEN
           runPhase(runEngine);
           resetQuestion(cmdRun2ph);
      END_IF;

      IF runEngine.top AND NOT filling.start THEN
           askQuestion(cmdRun3ph);
      END_IF;

      IF cmdRun3ph.answer = _Answers.ANS_YES THEN
           runPhase(filling);
           resetQuestion(cmdRun3ph);
      END_IF;

      IF filling.top THEN
            waitReset(IN:=TRUE, PT:= T#2S);
      END_IF;

      IF waitReset.Q THEN

          IF Im.kran6.onStatus = _statusDualInput.STATUS_On THEN
  	algManager.nMode:= ModeGpa.MODE_WORK_Ring;
          END_IF;
          IF Im.kran6.onStatus = _statusDualInput.STATUS_Off THEN
  	algManager.nMode:= ModeGpa.MODE_WORK_Line;
          END_IF;

          resetIfRunning(StrAlg);
      END_IF;

      StrAlg.isEnded:= filling.top;

  END_IF;

  StrAlg.CanRun := StrAlg.inCanRun;
  StrAlg.OpcCommandsDisabled := StrAlg.inOpcCommandsDisabled;

  (* ---- Если управление с ВУ заблокировано, то  передаем команду из алгоритма ---- *)
  IF StrAlg.inOpcCommandsDisabled THEN
  	StrAlg.inCommand := StrAlg.inCommand_Alg;
  ELSE (* иначе передаем команду с АРМа*)
  	StrAlg.inCommand := StrAlg.inCommand_ARM;
  END_IF;

  _sunpackerCommand(command := StrAlg.inCommand);
  	source := _sunpackerCommand.source;
  	cmd := _sunpackerCommand.cmd;

  IF cmd <> 0 AND lastCmd <> cmd AND (((NOT StrAlg.opcCommandsDisabled) AND source > 0) OR source = 0) then
  	CASE BYTE_TO_INT(cmd) OF
  		(*cmdRun*) 1: 	IF (StrAlg.CanRun) THEN
  					StrAlg.isRuning := TRUE;
  					StrAlg.isEnded := FALSE;
  					StrAlg.hasError := FALSE;
  					(*****************       OnRun       *****************)

                                                    algoritms.puskOilSystem.inCanRun:= TRUE	;
                                                    algoritms.filling.inCanRun:= TRUE	;
                                                    algoritms.engineRun.inCanRun:= TRUE	;

                                                    algManager.nMode:=ModeGpa.MODE_MPUSK;
                                                    (*impulseSO(Im.SingleOutputs.VzvodBREO);*)
                                                    askQuestion(cmdRun1ph);

  					cmd_for_Status := cmd;
  					source_for_Status := source;
  					command_error_for_Status := 0;
  				ELSE
  					StrAlg.isRuning := FALSE;
  					StrAlg.isEnded := FALSE;
  					StrAlg.hasError 	:= FALSE;

  					cmd_for_Status := 0;
  					source_for_Status := source;
  					command_error_for_Status := cmd;
  				END_IF;
  		(*cmdReset*) 2: 	StrAlg.isRuning := FALSE;
  				StrAlg.isEnded := FALSE;
  				StrAlg.hasError 	:= FALSE;

                                           (*****************       OnReset       *****************)
                                          waitReset(IN:=FALSE);
                                          StrAlg.inCanRun:=FALSE;

                                          resetPhase(runOilsystem);
                                          resetPhase(runEngine);
                                          resetPhase(filling);

                                          resetQuestion(cmdRun1ph);
                                          resetQuestion(cmdRun2ph);
                                          resetQuestion(cmdRun3ph);

                                          StrAlg.inOpcCommandsDisabled:=FALSE;

  				cmd_for_Status := cmd;
  				source_for_Status := source;
  				command_error_for_Status := 0;
  	END_CASE;
  	resetCmdTimer(IN := false);
  	resetCmdTimerPriznak := TRUE;
  END_IF;
  lastCmd := cmd;

  resetCmdTimer(IN := resetCmdTimerPriznak, PT := T#5S);
  IF resetCmdTimer.Q THEN
  	resetCmdTimerPriznak := FALSE;
  	source_for_Status := 0;
  	cmd_for_Status := 0;
  	command_error_for_Status := 0;
  END_IF;

  StrAlg.Start:= runOilsystem.startStatus
              OR runEngine.startStatus
              OR filling.startStatus;

  StrAlg.Error:= runOilsystem.errorStatus
              OR runEngine.errorStatus
              OR filling.errorStatus;

  StrAlg.Top:=   runOilsystem.topStatus
              OR runEngine.topStatus
              OR filling.topStatus;

  (*TODO: TYPE PROGRAM CODE HERE*)
  StrAlg.status :=  SHL(BYTE_TO_DWORD(source_for_Status), 29)
  			OR SHL(BYTE_TO_DWORD(cmd_for_Status), 26)
  			OR SHL(BYTE_TO_DWORD(command_error_for_Status), 23)
  			OR SHL(BOOL_TO_DWORD(StrAlg.OpcCommandsDisabled ), 21)
  			OR SHL(BOOL_TO_DWORD(StrAlg.hasError),4)
  			OR SHL(BOOL_TO_DWORD(StrAlg.CanRun),2)
  			OR SHL(BOOL_TO_DWORD(StrAlg.isEnded),1)
  			OR BOOL_TO_DWORD(StrAlg.isRuning);
END_FUNCTION_BLOCK

FUNCTION resetAllProtections : BOOL
  VAR_IN_OUT
    protections : ProtectionsConfig;
  END_VAR

  resetAiProtection(protections.Topornogo_podshipnika_EDT_1);
  resetAiProtection(protections.Toy_podshipnika_EDT_2);
  resetAiProtection(protections.Toy_podshipnika_kol_EDT_3);
  resetAiProtection(protections.Toy_podshipnika_kol_EDT_4);
  resetAiProtection(protections.To_podshipnika_shest_red_EDT_5);
  resetAiProtection(protections.To_podshipnika_shest_red_EDT_6);
  resetAiProtection(protections.To_podshipnika_N_EDT_7);
  resetAiProtection(protections.To_podshipnika_svob_konca_EDT_8);
  resetAiProtection(protections.Ty_podshipnika_rab_kol_EDT_9);
  resetAiProtection(protections.Typornogo_podshipnika_nerab_kolodok_HT_10);
  resetAiProtection(protections.Tgaza_na_vyhode_H);
  resetAiProtection(protections.Os_sdvig_nagnetatelja_plus);
  resetAiProtection(protections.Os_sdvig_nagnetatelja_minus);
  resetAiProtection(protections.Pgaza_na_vyhode_nagnetatelia_GPA_STOP);
  resetAiProtection(protections.Pgaza_na_vhode_nagnetatelia_GPA_STOP);
  resetAiProtection(protections.Pgaza_na_vyhode_nagnetatelia);
  resetAiProtection(protections.dPmaslo_gaz);
  resetAiProtection(protections.Pmaslo_sm_nizkoe);
  resetAiProtection(protections.Pmaslo_sm_vysokoe);
  resetAiProtection(protections.Vibro_skorost_OPED_T1);
  resetAiProtection(protections.Vibro_skorost_OPED_T2);
  resetAiProtection(protections.Vibro_skorost_OYP_kolesa_ED_T3);
  resetAiProtection(protections.Vibro_skorost_OP_kolesa_RH_T4);
  resetAiProtection(protections.Vibro_skorost_OP_shesterni_RED_T5);
  resetAiProtection(protections.Vibro_skorost_OP_shesterni_RED_T6);

  resetDiProtection(protections.dPmaslo_gaz_less100);
  resetDiProtection(protections.Reg_vozb_off);
  resetDiProtection(protections.Fail_chastotnii_pusk);
  resetDiProtection(protections.Off_avar_vikluchatel);
  resetDiProtection(protections.AOKC_SHKC);
  resetDiProtection(protections.AO_PRU);
  resetDiProtection(protections.AO_ot_SHU);
  resetDiProtection(protections.mvOff);
  resetDiProtection(protections.Kran1_sdvig);
  resetDiProtection(protections.Reg_vozb_off);
  resetDiProtection(protections.Kran2_sdvig);
END_FUNCTION

FUNCTION_BLOCK RemontAlg
  VAR_IN_OUT
    StrAlg : struct_Alg;
  END_VAR
  VAR
    _sunpackerCommand : fb_sunpackerCommand;
    source : BYTE;
    cmd : BYTE;
    lastCmd : BYTE;
    source_for_Status : BYTE;
    cmd_for_Status : BYTE;
    command_error_for_Status : BYTE;
    resetCmdTimer : TON;
    resetCmdTimerPriznak : BOOL;
  END_VAR
  VAR_EXTERNAL
    protectManager : struct_ProtectionsManager;
    algManager : struct_AlgoritmsManager;
    ModeGpa : TYPE_ModeGpa;
    PMcommand : TYPE_CommandsPotectionsManager;
    IM : ImConfig;
  END_VAR

  StrAlg.CanRun := StrAlg.inCanRun;
  StrAlg.OpcCommandsDisabled := StrAlg.inOpcCommandsDisabled;

  (* ---- Если управление с ВУ заблокировано, то передаем команду из алгоритма ---- *)
  IF StrAlg.inOpcCommandsDisabled THEN
  	StrAlg.inCommand := StrAlg.inCommand_Alg;
  ELSE (* иначе передаем команду с АРМа*)
  	StrAlg.inCommand := StrAlg.inCommand_ARM;
  END_IF;

  _sunpackerCommand(command := StrAlg.inCommand);
  	source := _sunpackerCommand.source;
  	cmd := _sunpackerCommand.cmd;

  IF cmd <> 0 AND lastCmd <> cmd AND (((NOT StrAlg.opcCommandsDisabled) AND source > 0) OR source = 0) then
  	CASE BYTE_TO_INT(cmd) OF
  		(*cmdRun*) 1: 	IF (StrAlg.CanRun) THEN
  					StrAlg.isRuning := TRUE;
  					StrAlg.isEnded := FALSE;
  					StrAlg.hasError 	:= FALSE;
                                               (*****************       OnRun       *****************)
                                                        algManager.nMode:=ModeGpa.MODE_REMONT;
                                                        protectManager.inCommand:=PMcommand.ResetAllProtections;
  					    UnBlockAllIM(IM);
                                                    (*StrAlg.inOpcCommandsDisabled:=FALSE;*)
  					cmd_for_Status := cmd;
  					source_for_Status := source;
  					command_error_for_Status := 0;
  				ELSE
  					StrAlg.isRuning := FALSE;
  					StrAlg.isEnded := FALSE;
  					StrAlg.hasError 	:= FALSE;

  					cmd_for_Status := 0;
  					source_for_Status := source;
  					command_error_for_Status := cmd;
  				END_IF;
  		(*cmdReset*) 2: 	StrAlg.isRuning := FALSE;
  				StrAlg.isEnded := FALSE;
  				StrAlg.hasError 	:= FALSE;
                                          (*****************       OnReset       *****************)
                                                    BlockAllIM(IM);
                                                    protectManager.inCommand:=PMcommand.RestartAllProtections;
                                                    algManager.nMode:=ModeGpa.MODE_STOP;

  				cmd_for_Status := cmd;
  				source_for_Status := source;
  				command_error_for_Status := 0;
  	END_CASE;
  	resetCmdTimer(IN := false);
  	resetCmdTimerPriznak := TRUE;
  END_IF;
  lastCmd := cmd;

  resetCmdTimer(IN := resetCmdTimerPriznak, PT := T#5S);
  IF resetCmdTimer.Q THEN
  	resetCmdTimerPriznak := FALSE;
  	source_for_Status := 0;
  	cmd_for_Status := 0;
  	command_error_for_Status := 0;
  END_IF;

  StrAlg.status :=  SHL(BYTE_TO_DWORD(source_for_Status), 29)
  			OR SHL(BYTE_TO_DWORD(cmd_for_Status), 26)
  			OR SHL(BYTE_TO_DWORD(command_error_for_Status), 23)
  			OR SHL(BOOL_TO_DWORD(StrAlg.OpcCommandsDisabled ), 21)
  			OR SHL(BOOL_TO_DWORD(StrAlg.hasError),4)
  			OR SHL(BOOL_TO_DWORD(StrAlg.CanRun),2)
  			OR SHL(BOOL_TO_DWORD(StrAlg.isEnded),1)
  			OR BOOL_TO_DWORD(StrAlg.isRuning);
END_FUNCTION_BLOCK

FUNCTION_BLOCK fb_SectionSwitch
  VAR_INPUT
    statOn : BOOL;
    statOff : BOOL;
    statOn_reliability : BOOL;
    statOff_reliability : BOOL;
  END_VAR
  VAR_IN_OUT
    StrSw : struct_SectionSwitch;
  END_VAR
  VAR_INPUT
    basketRolledIn : TYPE_ReliableBit;
    basketRolledOut : TYPE_ReliableBit;
    basketTest : TYPE_ReliableBit;
    inNs : TYPE_ReliableBit;
    inoffKNA : TYPE_ReliableBit;
    inAccident : TYPE_ReliableBit;
    inLocal : TYPE_ReliableBit;
    inDistance : TYPE_ReliableBit;
    inBreakCmdOn : TYPE_ReliableBit;
    inBreakCmdOff : TYPE_ReliableBit;
  END_VAR
  VAR
    onInit : BOOL          := FALSE;
    _statOn : BOOL;
    _statOff : BOOL;
    getSdvig : BOOL;
    lastOnStatus : BYTE;
    cmd : BYTE;
    source : BYTE;
    lastCmd : BYTE;
    source_for_Status : BYTE;
    cmd_for_Status : BYTE;
    command_error_for_Status : BYTE;
    _basketRolledIn : TYPE_ReliableBit;
    _basketRolledOut : TYPE_ReliableBit;
    _basketTest : TYPE_ReliableBit;
    _sunpackerCommand : fb_sunpackerCommand;
    _statusDualInput : TYPE_statusDualInput;
    _statusBasket : TYPE_basketStats;
    _commandDualInput : TYPE_commandDualInput;
    _commandErrorTimer : BOOL;
    resetErrorTimer : BOOL;
    _changWithoutCommand : BOOL;
    errorCMDTimer : TON;
    _errorReset : TON;
    sdvigReset : TON;
    outputsSets : TOF;
  END_VAR
  VAR_IN_OUT
    cmdOn : BOOL;
    cmdOff : BOOL;
  END_VAR

  IF NOT onInit THEN
  IF StrSw.ISVALIDREF_cmdOn XOR StrSw.ISVALIDREF_cmdOff THEN
  	IF 	StrSw.ISVALIDREF_cmdOn THEN
  		lastCmd:= 2; (*baseCmdOff*)
  	ELSE
  		lastCmd:= 1; (*baseCmdOn*)
  	END_IF;
  END_IF;
  onInit:=TRUE;
  END_IF;

  (* ---- Формирование состояния тележки ---- *)

  IF (NOT StrSw.ISVALIDREF_basketRolledIn) AND (NOT StrSw.ISVALIDREF_basketRolledOut) THEN
            StrSw.basketStatus:=_statusBasket.BASKET_NOTDEFINED;
  ELSE
  		IF StrSw.ISVALIDREF_basketTest THEN
  		_basketTest:=basketTest;
  	ELSE
  		_basketTest.reliability:=TRUE;
  		_basketTest.value :=FALSE;
  	END_IF;

  	IF StrSw.ISVALIDREF_basketRolledIn THEN
  		_basketRolledIn:=basketRolledIn;
  	ELSE
  		_basketRolledIn:=basketRolledOut;
  		IF StrSw.ISVALIDREF_basketTest THEN
  		_basketRolledIn.value:=NOT (_basketRolledIn.value OR _basketTest.value);
  		ELSE
  		_basketRolledIn.value:= NOT _basketRolledIn.value;
  		END_IF;

  	END_IF;

  	IF StrSw.ISVALIDREF_basketRolledOut THEN
  		_basketRolledOut:=basketRolledOut;
  	ELSE
  		_basketRolledOut:=basketRolledIn;
  		IF StrSw.ISVALIDREF_basketTest THEN
  		_basketRolledOut.value:= NOT (_basketRolledOut.value OR _basketTest.value );
  		ELSE
  			_basketRolledOut.value := NOT _basketRolledout.value;
  		END_IF;

  	END_IF;

  IF _basketRolledIn.reliability AND _basketRolledOut.reliability AND _basketTest.reliability THEN
  		IF (BOOL_TO_INT(_basketRolledIn.value)+BOOL_TO_INT(_basketRolledOut.value)+BOOL_TO_INT(_basketTest.value))=1 THEN
  			IF _basketRolledIn.value THEN
  				StrSw.basketStatus:=_statusBasket.BASKET_ROLLEDIN;
  			ELSIF _basketRolledOut.value THEN
  				StrSw.basketStatus:=_statusBasket.BASKET_ROLLEDOUT;
  			ELSIF _basketTest.value THEN
  				StrSw.basketStatus:=_statusBasket.BASKET_TEST;
  			END_IF;
  		ELSE
  			StrSw.basketStatus:=_statusBasket.BASKET_ERROR;
  		END_IF;
  	ELSE
  		StrSw.basketStatus:=_statusBasket.BASKET_NOTDEFINED;
  	END_IF;
  END_IF;

  (* ---- Если управление с ВУ заблокировано, то в ИМ передаем команду из алгоритма ---- *)
  IF StrSw.inOpcCommandsDisabled THEN
  	StrSw.inCommand := StrSw.inCommand_Alg;
  ELSE (* иначе передаем команду с АРМа*)
  	StrSw.inCommand := StrSw.inCommand_ARM;
  END_IF;

  (* ---- Формирование состояния механизма ---- *)

  IF (StrSw.ISVALIDREF_statOn) OR (StrSw.ISVALIDREF_statOff) THEN
  	IF (StrSw.ISVALIDREF_statOn) AND (StrSw.ISVALIDREF_statOff) THEN
  	StrSw.reliability:= statOn_reliability AND statOff_reliability;
  		_statOn  := statOn;
  		_statOff := statOff;
  	ELSIF (StrSw.ISVALIDREF_statOn) THEN
                       StrSw.reliability:= statOn_reliability;
  		_statOn  := statOn;
  		_statOff := NOT statOn;
  	ELSIF (StrSw.ISVALIDREF_statOff) THEN
  		 StrSw.reliability:= statOff_reliability;
  		_statOn  := NOT statOff;
  		_statOff :=statOff;
  	END_IF;

  	IF StrSw.reliability THEN
  		IF _statOn AND NOT _statOff 		THEN 	StrSw.onStatus := _statusDualInput.STATUS_ON;
  		ELSIF _statOff AND NOT _statOn 	THEN 	StrSw.onStatus := _statusDualInput.Status_OFF;
  		ELSIF NOT _statOn AND NOT _statOff 	THEN 	StrSw.onStatus := _statusDualInput.STATUS_TRANSITIONAL;
  		ELSE					StrSw.onStatus := _statusDualInput.STATUS_ERROR;
                      END_IF;

  	ELSE
  		StrSw.onStatus := _statusDualInput.STATUS_NOTDEFINED;

  	END_IF;
  ELSE
  	CASE BYTE_TO_INT(lastCmd) OF
  		(*baseCmdOn*) 1: StrSw.onStatus  := _statusDualInput.STATUS_ON;
  		(*baseCmdOff*) 2: StrSw.onStatus  := _statusDualInput.STATUS_OFF;

  	ELSE
  		 StrSw.onStatus := _statusDualInput.STATUS_NOTDEFINED;

  	END_CASE;
  END_IF;

  StrSw.Accident := inAccident.value AND inAccident.reliability;
  StrSw.Ns := inNs.value AND inNs.reliability;
  StrSw.Local := inLocal.value AND inLocal.reliability;
  StrSw.Distance := inDistance.value AND inDistance.reliability;
  StrSw.OpcCommandsDisabled := StrSw.inOpcCommandsDisabled;
  StrSw.offKNA := inoffKNA.value AND inoffKNA.reliability;

  (* ---- Формирование признака сдвига ---- *)

  getSdvig := FALSE;
  IF (StrSw.ISVALIDREF_cmdOn OR StrSw.ISVALIDREF_cmdOff) AND NOT StrSw.Local THEN
  	IF NOT (StrSw.CmdOn OR StrSw.CmdOff) THEN
                       IF (lastOnStatus <> StrSw.onStatus AND
  		(StrSw.onStatus <> _statusDualInput.STATUS_NOTDEFINED AND
                       StrSw.onStatus <> _statusDualInput.STATUS_ERROR)     AND
  		(lastOnStatus <> _statusDualInput.STATUS_NOTDEFINED   AND
                       lastOnStatus <> _statusDualInput.STATUS_ERROR))
                      THEN
  			getSdvig   := TRUE;
  		END_IF;
  	END_IF;
  END_IF;

  IF getSdvig THEN StrSw.sdvig:= TRUE; END_IF;

  sdvigReset(IN:=StrSw.sdvig, PT:=T#15S);

  IF sdvigReset.Q THEN StrSw.sdvig:=FALSE; END_IF;

  lastOnStatus := StrSw.onStatus;

  (* ---- Распаковка команды ---- *)
  _sunpackerCommand(command := StrSw.inCommand);
  	cmd := _sunpackerCommand.cmd;
  	source := _sunpackerCommand.source;

  (* ---- Обработка команды ---- *)
  IF cmd <> 0 AND lastCmd <> cmd and (((NOT StrSw.opcCommandsDisabled) AND source > 0) OR source = 0) then
  	CASE BYTE_TO_INT(cmd) OF
  	(*cmd_open*) 1 :
  			IF  StrSw.ISVALIDREF_cmdOn THEN StrSw.CmdOn := TRUE;
  				IF StrSw.ISVALIDREF_cmdOff THEN StrSw.CmdOff := FALSE; END_IF;
  			ELSIF  StrSw.ISVALIDREF_cmdOff THEN StrSw.CmdOff := FALSE;  END_IF;
  			errorCMDTimer(IN := false);
  			_commandErrorTimer := true;
  			StrSw.lastCmdIsOn := true;
  	(*cmd_close*) 2 :
  			IF StrSw.ISVALIDREF_cmdOff THEN StrSw.CmdOff := TRUE;
  				IF StrSw.ISVALIDREF_cmdOn THEN StrSw.CmdOn := FALSE; END_IF;
  			ELSIF StrSw.ISVALIDREF_cmdOn THEN StrSw.CmdOn := FALSE; END_IF;
  			errorCMDTimer(IN := false);
  			_commandErrorTimer := true;
  			StrSw.lastCmdIsOn := false;
  	(*cmd_reset*) 3 :    IF StrSw.ISVALIDREF_statOn OR StrSw.ISVALIDREF_statOff THEN
  			StrSw.CmdOn := FALSE;
  			StrSw.CmdOff := FALSE;
                                lastCmd := 0;
  			_commandErrorTimer := false;
  			StrSw.lastCmdIsOn := false;
                                 END_IF;
  	END_CASE;
  	source_for_Status := source;
  	cmd_for_Status := cmd;
  	command_error_for_Status := 0;
  END_IF;
  lastCmd := cmd;

  errorCMDTimer(In := _commandErrorTimer, PT :=T#10s);

  (* ---- алгоритм  для команды ВКЛючить ---- *)
  IF (StrSw.onStatus = _statusDualInput.STATUS_ON) and (StrSw.lastCmdIsOn) then
  	IF StrSw.ISVALIDREF_cmdOn AND StrSw.ISVALIDREF_cmdOff then  StrSw.cmdOn := false; END_IF;

  	 errorCMDTimer(In := false);
  	 _commandErrorTimer := false;
  	 cmd_for_Status := 0;
  	 source_for_Status := 0;
  END_IF;

  (* ---- off ---- *)
  IF (StrSw.onStatus = _statusDualInput.STATUS_OFF) and (NOT StrSw.lastCmdIsOn) then
  	IF StrSw.ISVALIDREF_cmdOn AND StrSw.ISVALIDREF_cmdOff then  StrSw.cmdOff := false; END_IF;

  	 errorCMDTimer(In := false);
  	 _commandErrorTimer := false;
  	 cmd_for_Status := 0;
  	 source_for_Status := 0;
  END_IF;

  (* ---- ошибка исполнения команды ---- *)
  if errorCMDTimer.Q and (cmd_for_Status <> 0) then
  	command_error_for_Status :=  cmd_for_Status;
  	_commandErrorTimer := false;
  	StrSw.CmdOn := false;
  	StrSw.CmdOff := false;
  	lastCmd := 0;
  end_if;

  (* ---- сброс ошибки команды ---- *)
  StrSw.CommandFault := command_error_for_Status <> 0;
  _errorReset(IN := command_error_for_Status <> 0, PT := T#5S);
  IF _errorReset.Q THEN
  	cmd_for_Status := 0;
  	source_for_Status := 0;
  	command_error_for_Status := 0;
  END_IF;

  outputsSets(in := (StrSw.ISVALIDREF_cmdOn and StrSw.cmdOn ) OR (StrSw.ISVALIDREF_cmdOff and StrSw.cmdOff), PT := T#2S);
  	IF NOT outputsSets.Q THEN
  		StrSw.BreakCmdOn := inBreakCmdOn._inversed AND inBreakCmdOn.reliability AND StrSw.ISVALIDREF_inBreakCmdOn;
  		StrSw.BreakCmdOff := inBreakCmdOff._inversed AND inBreakCmdOff.reliability AND StrSw.ISVALIDREF_inBreakCmdOff;
  	END_IF;

  cmdOn := StrSw.cmdOn;
  cmdOff:= StrSw.cmdOff;

  (* ---- формирование зашифрованного статуса для АРМа ---- *)
  StrSw.status := shl(BYTE_TO_DWORD(source_for_Status), 29)
  		OR shl(BYTE_TO_DWORD(cmd_for_Status), 26)
  		OR shl(BYTE_TO_DWORD(command_error_for_Status), 23)
  		OR shl(bool_to_DWORD(StrSw.sdvig), 22)
  		OR shl(bool_to_DWORD(StrSw.OpcCommandsDisabled), 21)
                      OR shl(BOOL_TO_DWORD(StrSw.offKNA), 17)
                      OR shl(bool_to_DWORD(StrSw.lastCmdIsOn), 14)
                      OR shl(BOOL_TO_DWORD(StrSw.BreakCmdOff), 13)
  		OR shl(BOOL_TO_DWORD(StrSw.BreakCmdOn), 12)
                      OR shl(BYTE_TO_DWORD(StrSw.basketStatus), 8)
  		OR shl(BOOL_TO_DWORD(StrSw.Distance), 6)
  		OR shl(BOOL_TO_DWORD(StrSw.Local), 5)
  		OR shl(BOOL_TO_DWORD(StrSw.Ns), 4)
                  	OR shl(BOOL_TO_DWORD(StrSw.Accident ),3)
  		OR BYTE_TO_DWORD(StrSw.onStatus);
END_FUNCTION_BLOCK

FUNCTION_BLOCK fb_DiscretParametr
  VAR_IN_OUT
    StrDP : struct_DiscretParametr;
  END_VAR
  VAR
    _sunpackerCommand : fb_sunpackerCommand;
    source : BYTE;
    cmd : BYTE;
    parametr : BYTE;
    lastParametr : BYTE;
    source_for_Status : BYTE;
    cmd_for_Status : BYTE;
    command_error_for_Status : BYTE;
    resetCmdTimer : TON;
    resetCmdTimerPriznak : BOOL;
    secondTact : BOOL;
  END_VAR

  IF NOT secondTact THEN
  	StrDP.Value := StrDP.currentValue;
  	secondTact := true;
  END_IF;

  StrDP.OpcCommandsDisabled := StrDP.inOpcCommandsDisabled;

  (* ---- Если управление с ВУ заблокировано, то передаем команду из алгоритма ---- *)
  IF StrDP.inOpcCommandsDisabled THEN
  	StrDP.inCommand := StrDP.inCommand_Alg;
  ELSE (* иначе передаем команду с АРМа*)
  	StrDP.inCommand := StrDP.inCommand_ARM;
  END_IF;

  _sunpackerCommand(command := StrDP.inCommand);
  	source := _sunpackerCommand.source;
            parametr := _sunpackerCommand.parametr;
  	cmd := _sunpackerCommand.cmd;

  IF NOT StrDP.inOpcCommandsDisabled THEN
  StrDP.newValue:= BYTE_TO_UINT(parametr);
  END_IF;

  IF cmd <> 0 AND StrDP.Value <> StrDP.newValue AND (((NOT StrDP.opcCommandsDisabled) AND source > 0) OR source = 0) then
  	CASE BYTE_TO_INT(cmd) OF
  	(*cmd_ChangeValue*) 1 :
                                    StrDP.Value := StrDP.newValue;
                                    StrDP.opcCommandsDisabled:=FALSE;
  	END_CASE;
  	source_for_Status := source;
  	cmd_for_Status := cmd;
  	resetCmdTimer(IN := FALSE);
  	resetCmdTimerPriznak := TRUE;
  END_IF;

  lastParametr := parametr;

  StrDP.status := SHL(BYTE_TO_DWORD(source_for_Status), 29)
  			OR SHL(BYTE_TO_DWORD(cmd_for_Status), 26)
  			OR SHL(BYTE_TO_DWORD(command_error_for_Status), 23)
  			OR SHL(BOOL_TO_DWORD(StrDP.OpcCommandsDisabled ), 21)
                                OR SHL(UINT_TO_DWORD(StrDP.Value), 5);

  resetCmdTimer(IN := resetCmdTimerPriznak, PT := T#5S);
  IF resetCmdTimer.Q THEN
  	resetCmdTimerPriznak := FALSE;
  	source_for_Status := 0;
  	cmd_for_Status := 0;
  	command_error_for_Status := 0;
  END_IF;
END_FUNCTION_BLOCK

FUNCTION_BLOCK fb_DiProtection_Init
  VAR_INPUT
    data_Ini : BOOL;
    delay : TIME;
    inTag : BYTE;
    inRunOnStart : BOOL;
  END_VAR
  VAR_IN_OUT
    str_DIp : struct_DiProtection;
  END_VAR
  VAR_OUTPUT
    Init : BOOL          := FALSE;
  END_VAR

  (*****            Функциональный блок переинициализации структуры  AiProtection          *****)

   Init := FALSE;

      IF data_Ini THEN                            (* Параметрам требуется переинициализация. *)
          str_DIp.delay               := delay;
          str_DIp.inTag               := inTag;
          str_DIp.inRunOnStart        := inRunOnStart;

          data_Ini:=FALSE;
          Init := TRUE;
      END_IF;
      IF Init THEN
          delay:= T#0S;
          inTag:= 0;
          inRunOnStart:= FALSE;
      END_IF;
END_FUNCTION_BLOCK

FUNCTION_BLOCK Pusk_first_faza2
  VAR_IN_OUT
    StrAlg : struct_Alg;
  END_VAR
  VAR
    nu1On : struct_PhaseAlgoritm;
    nu2On : struct_PhaseAlgoritm;
    timer240 : struct_PhaseAlgoritm;
    dPmg_more100 : struct_PhaseAlgoritm;
    Auto_NU1 : struct_PhaseAlgoritm;
    Error_Alg : struct_PhaseAlgoritm;
    fb_timer240 : fb_ph_Timer;
    fb_nu1On : fb_ph_OilPump;
    fb_nu2On : fb_ph_OilPump;
    fb_dPmg_more100 : fb_ph_algoritm;
    fb_Auto_NU1 : fb_ph_algoritm;
    fb_Error_Alg : fb_ph_algoritm;
    _sunpackerCommand : fb_sunpackerCommand;
    _statusDualInput : TYPE_statusDualInput;
    _Answers : TYPE_Answers;
    source : BYTE;
    cmd : BYTE;
    lastCmd : BYTE;
    source_for_Status : BYTE;
    cmd_for_Status : BYTE;
    command_error_for_Status : BYTE;
    resetCmdTimer : TON;
    resetCmdTimerPriznak : BOOL;
    onInit : BOOL;
    waitReset : TON;
  END_VAR
  VAR_EXTERNAL
    ModeGpa : TYPE_ModeGpa;
    algManager : struct_AlgoritmsManager;
    IM : ImConfig;
    protections : ProtectionsConfig;
    algoritms : AlgoritmsConfig;
    ai : AiConfig;
  END_VAR
  VAR
    statusAi : TYPE_StatusAi;
  END_VAR

  IF NOT onInit THEN
           fb_nu1On(phaseNumber:=1, act:=_on );
           fb_nu2On(phaseNumber:=2, act:=_on);
           fb_dPmg_more100(phaseNumber:=3);
           fb_Error_Alg(phaseNumber:=4);
           fb_Auto_NU1(phaseNumber:=5);
  onInit:=TRUE;
  END_IF;

  fb_timer240(StrPh:=timer240);
  fb_nu1On(StrPh:= nu1On,Im:=Im.nu1);
  fb_nu2On(StrPh:= nu2On,Im:=Im.nu2);
  fb_dPmg_more100(StrPh:=dPmg_more100);
  fb_Auto_NU1(StrPh:=Auto_NU1, alg:=algoritms.autoNu); (*komu ono nujno to blat *)
  fb_Error_Alg(StrPh:=Error_Alg);

  StrAlg.CanRun := StrAlg.inCanRun;
  StrAlg.OpcCommandsDisabled := StrAlg.inOpcCommandsDisabled;

  IF StrAlg.isRuning THEN

      StrAlg.hasError := nu1On.error AND nu2On.error AND Auto_NU1.error;

      (* защита не возведена - запускаем таймер *)
      IF NOT dPmg_more100.top THEN
  	runPhase(timer240);
      END_IF;

      (* носос 1 не включен - включаем насос*)
      IF NOT nu1On.start THEN
  	runPhase(nu1On);
      END_IF;

      (* носос 2 не включен - включаем насос*)
      IF NOT nu2On.start THEN
  	runPhase(nu2On);
      END_IF;

      (* один из насосов включен - включение защиты *)
      IF ((IM.nu1.onStatus = _statusDualInput.status_on OR IM.nu2.onStatus = _statusDualInput.status_on) AND  (nu1On.start OR nu2On.Start)) THEN
  	runPhase(dPmg_more100);
  	nu1On.top:=TRUE;
            nu2On.top:=TRUE;
      END_IF;

      (* фаза защиты активна - включение защиты *)
      IF dPmg_more100.start AND NOT dPmg_more100.top THEN
  	IF NOT IM.SingleSignals.dP_maslo_gaz_Less100.Q AND IM.SingleSignals.dP_maslo_gaz_Less100.status = 1 AND
  	ai.dPmaslo_gaz.interval >= statusAi.normal AND ai.dPmaslo_gaz.value > 150.0 THEN
                dPmg_more100.top:=TRUE;
  	END_IF;
      END_IF;

      (*таймер завершился до возведения защит - ошибка *)
      IF timer240.top THEN
  	Error_Alg.error := TRUE;
      ELSE
  	Error_Alg.error := FALSE;
      END_IF;

      IF dPmg_more100.top AND nu1On.top AND nu2On.top THEN
  	Auto_NU1.top:=TRUE;
  	runAiProtection(protections.dPmaslo_gaz);
            runDiProtection(protections.dPmaslo_gaz_less100);
  	resetAiProtection(protections.Pgaza_na_vhode_nagnetatelia_GPA_STOP);
  	resetAiProtection(protections.Pgaza_na_vyhode_nagnetatelia_GPA_STOP);
  	algoritms.autoNu.CanRun:=TRUE;
  	(*algoritms.autoNu.run ();ниче не ясно*)
  	resetPhase(timer240);
      END_IF;
  END_IF;

  StrAlg.CanRun := StrAlg.inCanRun;
  StrAlg.OpcCommandsDisabled := StrAlg.inOpcCommandsDisabled;

  (* ---- Если управление с ВУ заблокировано, то  передаем команду из алгоритма ---- *)
  IF StrAlg.inOpcCommandsDisabled THEN
  	StrAlg.inCommand := StrAlg.inCommand_Alg;
  ELSE (* иначе передаем команду с АРМа*)
  	StrAlg.inCommand := StrAlg.inCommand_ARM;
  END_IF;

  _sunpackerCommand(command := StrAlg.inCommand);
  	source := _sunpackerCommand.source;
  	cmd := _sunpackerCommand.cmd;

  IF cmd <> 0 AND lastCmd <> cmd AND (((NOT StrAlg.opcCommandsDisabled) AND source > 0) OR source = 0) then
  	CASE BYTE_TO_INT(cmd) OF
  		(*cmdRun*) 1: 	IF (StrAlg.CanRun) THEN
  					StrAlg.isRuning := TRUE;
  					StrAlg.isEnded := FALSE;
  					StrAlg.hasError := FALSE;
  					(*****************       OnRun       *****************)
                                                    algManager.nMode:=ModeGpa.MODE_PUSK_FIRST_FAZA2;

                                                    runPhase(timer240);
                                                    runPhase(nu1On);
                                                    runPhase(nu2On);
                                                    resetAiProtection(protections.dPmaslo_gaz);
                                                    resetDiProtection(protections.dPmaslo_gaz_less100);

  					cmd_for_Status := cmd;
  					source_for_Status := source;
  					command_error_for_Status := 0;
  				ELSE
  					StrAlg.isRuning := FALSE;
  					StrAlg.isEnded := FALSE;
  					StrAlg.hasError := FALSE;

  					cmd_for_Status := 0;
  					source_for_Status := source;
  					command_error_for_Status := cmd;
  				END_IF;
  		(*cmdReset*) 2: 	StrAlg.isRuning := FALSE;
  				StrAlg.isEnded := FALSE;
  				StrAlg.hasError 	:= FALSE;

                                           (*****************       OnReset       *****************)
                                          waitReset(IN:=FALSE);
                                          StrAlg.inCanRun:=FALSE;

                                          resetPhase(nu1On);
                                          resetPhase(nu2On);
                                          resetPhase(timer240);
                                          resetPhase(dPmg_more100);
                                          resetPhase(Auto_NU1);
                                          resetPhase(Error_Alg);

                                          StrAlg.inOpcCommandsDisabled:=FALSE;

  				cmd_for_Status := cmd;
  				source_for_Status := source;
  				command_error_for_Status := 0;
  	END_CASE;
  	resetCmdTimer(IN := false);
  	resetCmdTimerPriznak := TRUE;
  END_IF;
  lastCmd := cmd;

  resetCmdTimer(IN := resetCmdTimerPriznak, PT := T#5S);
  IF resetCmdTimer.Q THEN
  	resetCmdTimerPriznak := FALSE;
  	source_for_Status := 0;
  	cmd_for_Status := 0;
  	command_error_for_Status := 0;
  END_IF;

  StrAlg.Start:= timer240.startStatus
              OR nu1On.startStatus
              OR nu2On.startStatus
              OR dPmg_more100.startStatus
              OR Auto_NU1.startStatus
              OR Error_Alg.startStatus;

  StrAlg.Error := timer240.errorStatus
              OR nu1On.errorStatus
              OR nu2On.errorStatus
              OR dPmg_more100.errorStatus
              OR Auto_NU1.errorStatus
              OR Error_Alg.errorStatus;

  StrAlg.Top := timer240.topStatus
              OR nu1On.topStatus
              OR nu2On.topStatus
              OR dPmg_more100.topStatus
              OR Auto_NU1.topStatus
              OR Error_Alg.topStatus;

  (*TODO: TYPE PROGRAM CODE HERE*)
  StrAlg.status :=  SHL(BYTE_TO_DWORD(source_for_Status), 29)
  			OR SHL(BYTE_TO_DWORD(cmd_for_Status), 26)
  			OR SHL(BYTE_TO_DWORD(command_error_for_Status), 23)
  			OR SHL(BOOL_TO_DWORD(StrAlg.OpcCommandsDisabled ), 21)
  			OR SHL(BOOL_TO_DWORD(StrAlg.hasError),4)
  			OR SHL(BOOL_TO_DWORD(StrAlg.CanRun),2)
  			OR SHL(BOOL_TO_DWORD(StrAlg.isEnded),1)
  			OR BOOL_TO_DWORD(StrAlg.isRuning);
END_FUNCTION_BLOCK

FUNCTION_BLOCK Pusk_third_faza
  VAR_IN_OUT
    StrAlg : struct_Alg;
  END_VAR
  VAR
    timer480 : struct_PhaseAlgoritm;
    kran4Open : struct_PhaseAlgoritm;
    waitAfterKran4 : struct_PhaseAlgoritm;
    kran5Close : struct_PhaseAlgoritm;
    kran3bOpen : struct_PhaseAlgoritm;
    dP_kr1less100 : struct_PhaseAlgoritm;
    Pvh_vyhMore5 : struct_PhaseAlgoritm;
    kran1Open : struct_PhaseAlgoritm;
    kran2Open : struct_PhaseAlgoritm;
    kran3Open : struct_PhaseAlgoritm;
    kran3bClose : struct_PhaseAlgoritm;
    Err_ALG : struct_PhaseAlgoritm;
    fb_timer480 : fb_ph_Timer;
    fb_kran4Open : fb_ph_Kran;
    fb_waitAfterKran4 : fb_ph_Timer;
    fb_kran5Close : fb_ph_Kran;
    fb_kran3bOpen : fb_ph_Kran;
    fb_dP_kr1less100 : fb_ph_algoritm;
    fb_Pvh_vyhMore5 : fb_ph_algoritm;
    fb_kran1Open : fb_ph_Kran;
    fb_kran2Open : fb_ph_Kran;
    fb_kran3Open : fb_ph_Kran;
    fb_kran3bClose : fb_ph_Kran;
    fb_Err_ALG : fb_ph_algoritm;
    _sunpackerCommand : fb_sunpackerCommand;
    _statusDualInput : TYPE_statusDualInput;
    _Answers : TYPE_Answers;
    source : BYTE;
    cmd : BYTE;
    lastCmd : BYTE;
    source_for_Status : BYTE;
    cmd_for_Status : BYTE;
    command_error_for_Status : BYTE;
    resetCmdTimer : TON;
    resetCmdTimerPriznak : BOOL;
    onInit : BOOL;
    waitReset : TON;
  END_VAR
  VAR_EXTERNAL
    ModeGpa : TYPE_ModeGpa;
    algManager : struct_AlgoritmsManager;
    IM : ImConfig;
    protections : ProtectionsConfig;
    algoritms : AlgoritmsConfig;
    ai : AiConfig;
  END_VAR
  VAR
    statusAi : TYPE_StatusAi;
  END_VAR

  IF NOT onInit THEN
           fb_timer480(phaseNumber:=1, delay:=T#480S);
           fb_kran4Open(phaseNumber:=2, act:=_on);
           fb_waitAfterKran4(phaseNumber:=3, delay:=T#10S);
           fb_kran5Close(phaseNumber:=4, act:=_off);
           fb_kran3bOpen(phaseNumber:=5, act:=_on);
           fb_dP_kr1less100(phaseNumber:=6);
           fb_Pvh_vyhMore5(phaseNumber:=7);
           fb_kran1Open(phaseNumber:=8, act:=_on);
           fb_kran2Open(phaseNumber:=9, act:=_on);
           fb_kran3Open(phaseNumber:=10, act:=_on);
           fb_kran3bClose(phaseNumber:=11, act:=_off);
           fb_Err_ALG(phaseNumber:=12);
  onInit:=TRUE;
  END_IF;

  fb_timer480(StrPh:=timer480);
  fb_kran4Open(StrPh:= kran4Open, Im:=Im.kran4);
  fb_waitAfterKran4(StrPh:= waitAfterKran4);
  fb_kran5Close(StrPh:=kran5Close, Im:=Im.kran5);
  fb_kran3bOpen(StrPh:=kran3bOpen, Im:=Im.kran3b);
  fb_dP_kr1less100(StrPh:=dP_kr1less100);
  fb_Pvh_vyhMore5(StrPh:=Pvh_vyhMore5);
  fb_kran1Open(StrPh:=kran1Open, Im:=Im.kran1);
  fb_kran2Open(StrPh:=kran2Open, Im:=Im.kran2);
  fb_kran3Open(StrPh:=kran3Open, Im:=Im.kran3);
  fb_kran3bClose(StrPh:=kran3bClose, Im:=Im.kran3b);
  fb_Err_ALG(StrPh:=Err_ALG);

  StrAlg.CanRun := StrAlg.inCanRun;
  StrAlg.OpcCommandsDisabled := StrAlg.inOpcCommandsDisabled;

  IF StrAlg.isRuning THEN
      (* запуск таймера *)
      IF NOT (kran3bClose.top) THEN
  	    runPhase(timer480);
      END_IF;

      (*если кран1 не открыт - октрыть кран 4*)
      IF	NOT kran1Open.top (*AND IM.kran4._cmdreset.IN = FALSE*)  THEN
  	    runIfNotRunningSO(IM.SingleOutputs.Kr4_open_from_alg);
  	    runPhase(kran4Open);
      END_IF;
      IF	kran4Open.start AND NOT kran4Open.top THEN
  	    IF	IM.kran4.onStatus = _statusDualInput.STATUS_ON THEN
  		    kran4Open.top:=TRUE;
  	    END_IF;
      END_IF;

      (* продувка крана *)
      IF kran4Open.top THEN
          runPhase(waitAfterKran4);
      END_IF;

      (* кран продулся - закрытие кран 5*)
      IF waitAfterKran4.top THEN
  	    runPhase(kran5Close);
      END_IF;

      (* кран 5 закрыт - открытие крана 3б проверка перепада давление*)
      IF	kran5Close.top THEN
  	    runPhase(kran3bOpen);
  	    runPhase(dP_kr1less100);
  	    runPhase(Pvh_vyhMore5);
      END_IF;

      (* проверка давления крана *)
      IF	Pvh_vyhMore5.start AND NOT Pvh_vyhMore5.top THEN
  	    IF	(ai.Pgaza_na_vhode_nagnetatelia.interval >=statusAi.NORMAL) AND (ai.Pgaza_na_vhode_nagnetatelia.value	 >= 4.0) AND
  		    (ai.Pgaza_na_vyhode_nagnetatelia.interval >=statusAi.NORMAL) AND (ai.Pgaza_na_vyhode_nagnetatelia.value	 >= 4.0) THEN
  		        Pvh_vyhMore5.top := TRUE;
      		    runAiProtection(protections.Pgaza_na_vyhode_nagnetatelia);
  	    END_IF;
      END_IF;

      (* проверка открытия крана 3б *)
      IF	kran3bOpen.start AND NOT kran3bOpen.top THEN
  	    IF	IM.kran3b.onStatus=_statusDualInput.STATUS_ON THEN
  		    kran3bOpen.top :=TRUE;
  	    END_IF;
      END_IF;
      IF	kran3bOpen.top AND	kran5Close.top AND dP_kr1less100.top AND Pvh_vyhMore5.top THEN
  	    runPhase(kran1Open);
  	    runPhase(kran2Open);
  	    runPhase(kran3Open);
  	    (*Smazka_1_2:=TRUE; нет такого *)
      END_IF;
      IF	kran1Open.top THEN
  	    resetIfRunningSO(IM.SingleOutputs.Kr4_open_from_alg);
  	    (*ystavki.Block_kr4_alg.setValue (0);что такое уставки*)
      END_IF;

      (* закрытие крана 3бис *)
      IF kran1Open.top AND kran2Open.top AND kran3Open.top THEN
  	    runPhase(kran3bClose);
      END_IF;
      IF 	kran3bClose.top THEN
  	    Err_ALG.error :=FALSE;
  	    resetPhase(timer480);
      ELSIF NOT kran3bClose.top AND timer480.top THEN
  		Err_ALG.error :=TRUE;
      END_IF;
  END_IF;

  _sunpackerCommand(command := StrAlg.inCommand);
  	source := _sunpackerCommand.source;
  	cmd := _sunpackerCommand.cmd;

  IF cmd <> 0 AND lastCmd <> cmd AND (((NOT StrAlg.opcCommandsDisabled) AND source > 0) OR source = 0) then
  	CASE BYTE_TO_INT(cmd) OF
  		(*cmdRun*) 1: 	IF (StrAlg.CanRun) THEN
  					StrAlg.isRuning := TRUE;
  					StrAlg.isEnded := FALSE;
  					StrAlg.hasError := FALSE;
  					(*****************       OnRun       *****************)
                                                    algManager.nMode:=ModeGpa.MODE_PUSK_FIRST_FAZA2;

                                                    (*runPhase(timer120);
                                                    runPhase(timer5);
                                                    runPhase(Shup);
                                                    resetAiProtection(protections.dPmaslo_gaz);
                                                    resetDiProtection(protections.dPmaslo_gaz_less100);*)

  					cmd_for_Status := cmd;
  					source_for_Status := source;
  					command_error_for_Status := 0;
  				ELSE
  					StrAlg.isRuning := FALSE;
  					StrAlg.isEnded := FALSE;
  					StrAlg.hasError := FALSE;

  					cmd_for_Status := 0;
  					source_for_Status := source;
  					command_error_for_Status := cmd;
  				END_IF;
  		(*cmdReset*) 2: 	StrAlg.isRuning := FALSE;
  				StrAlg.isEnded := FALSE;
  				StrAlg.hasError 	:= FALSE;

                                           (*****************       OnReset       *****************)
                                          waitReset(IN:=FALSE);
                                          StrAlg.inCanRun:=FALSE;

                                          (*resetPhase(timer5);
                                          resetPhase(Shup);
                                          resetPhase(timer120);
                                          resetPhase(Net_Chast);
                                          resetPhase(mvOn);
                                          resetPhase(pGNSmore04);
                                          resetPhase(gotov_K_zagruzke);
                                          resetPhase(dPmg_Top);
                                          resetPhase(AutoPNS_Start);*)

                                          StrAlg.inOpcCommandsDisabled:=FALSE;

  				cmd_for_Status := cmd;
  				source_for_Status := source;
  				command_error_for_Status := 0;
  	END_CASE;
  	resetCmdTimer(IN := false);
  	resetCmdTimerPriznak := TRUE;
  END_IF;
  lastCmd := cmd;

  resetCmdTimer(IN := resetCmdTimerPriznak, PT := T#5S);
  IF resetCmdTimer.Q THEN
  	resetCmdTimerPriznak := FALSE;
  	source_for_Status := 0;
  	cmd_for_Status := 0;
  	command_error_for_Status := 0;
  END_IF;

  StrAlg.Start:= timer480.startStatus
              OR kran4Open.startStatus
              OR waitAfterKran4.startStatus
              OR kran5Close.startStatus
              OR kran3bOpen.startStatus
              OR dP_kr1less100.startStatus
              OR Pvh_vyhMore5.startStatus
              OR kran1Open.startStatus
              OR kran2Open.startStatus
              OR kran3Open.startStatus
              OR kran3bClose.startStatus
              OR Err_ALG.startStatus;

  StrAlg.Error := timer480.errorStatus
              OR kran4Open.errorStatus
              OR waitAfterKran4.errorStatus
              OR kran5Close.errorStatus
              OR kran3bOpen.errorStatus
              OR dP_kr1less100.errorStatus
              OR Pvh_vyhMore5.errorStatus
              OR kran1Open.errorStatus
              OR kran2Open.errorStatus
              OR kran3Open.errorStatus
              OR kran3bClose.errorStatus
              OR Err_ALG.errorStatus;

  StrAlg.Top := timer480.topStatus
              OR kran4Open.topStatus
              OR waitAfterKran4.topStatus
              OR kran5Close.topStatus
              OR kran3bOpen.topStatus
              OR dP_kr1less100.topStatus
              OR Pvh_vyhMore5.topStatus
              OR kran1Open.topStatus
              OR kran2Open.topStatus
              OR kran3Open.topStatus
              OR kran3bClose.topStatus
              OR Err_ALG.topStatus;

  (*TODO: TYPE PROGRAM CODE HERE*)
  StrAlg.status :=  SHL(BYTE_TO_DWORD(source_for_Status), 29)
  			OR SHL(BYTE_TO_DWORD(cmd_for_Status), 26)
  			OR SHL(BYTE_TO_DWORD(command_error_for_Status), 23)
  			OR SHL(BOOL_TO_DWORD(StrAlg.OpcCommandsDisabled ), 21)
  			OR SHL(BOOL_TO_DWORD(StrAlg.hasError),4)
  			OR SHL(BOOL_TO_DWORD(StrAlg.CanRun),2)
  			OR SHL(BOOL_TO_DWORD(StrAlg.isEnded),1)
  			OR BOOL_TO_DWORD(StrAlg.isRuning);
END_FUNCTION_BLOCK

FUNCTION_BLOCK Pusk_second_faza_reactor
  VAR_IN_OUT
    StrAlg : struct_Alg;
  END_VAR
  VAR
    timer25 : struct_PhaseAlgoritm;
    timer3 : struct_PhaseAlgoritm;
    mvOn : struct_PhaseAlgoritm;
    pGNSmore04 : struct_PhaseAlgoritm;
    gotov_K_zagruzke : struct_PhaseAlgoritm;
    dPmg_Top : struct_PhaseAlgoritm;
    Mv_Error : struct_PhaseAlgoritm;
    AutoPNS_Start : struct_PhaseAlgoritm;
    fb_timer25 : fb_ph_Timer;
    fb_timer3 : fb_ph_Timer;
    fb_Mv_Error : fb_ph_algoritm;
    fb_mvOn : fb_ph_SectionSwitch;
    fb_pGNSmore04 : fb_ph_algoritm;
    fb_gotov_K_zagruzke : fb_ph_algoritm;
    fb_dPmg_Top : fb_ph_algoritm;
    fb_AutoPNS_Start : fb_ph_algoritm;
    _sunpackerCommand : fb_sunpackerCommand;
    _statusDualInput : TYPE_statusDualInput;
    _Answers : TYPE_Answers;
    source : BYTE;
    cmd : BYTE;
    lastCmd : BYTE;
    source_for_Status : BYTE;
    cmd_for_Status : BYTE;
    command_error_for_Status : BYTE;
    resetCmdTimer : TON;
    resetCmdTimerPriznak : BOOL;
    onInit : BOOL;
    waitReset : TON;
  END_VAR
  VAR_EXTERNAL
    ModeGpa : TYPE_ModeGpa;
    algManager : struct_AlgoritmsManager;
    IM : ImConfig;
    protections : ProtectionsConfig;
    algoritms : AlgoritmsConfig;
    ai : AiConfig;
  END_VAR
  VAR
    statusAi : TYPE_StatusAi;
  END_VAR

  IF NOT onInit THEN
           fb_timer25(phaseNumber:=1, delay:=T#25S);
           fb_timer3(phaseNumber:=2, delay:=T#3S);
           fb_mvOn(phaseNumber:=3, act:=_on);
           fb_pGNSmore04(phaseNumber:=4);
           fb_gotov_K_zagruzke(phaseNumber:=5);
           fb_dPmg_Top(phaseNumber:=6);
           fb_Mv_Error(phaseNumber:=7);
           fb_AutoPNS_start(phaseNumber:=8, act:=_run, waitCompletion:=FALSE);

  onInit:=TRUE;
  END_IF;

  fb_timer25(StrPh:=timer25);
  fb_timer3(StrPh:= timer3);
  fb_mvOn(StrPh:= mvOn, Im:=IM.mv);
  fb_pGNSmore04(StrPh:=pGNSmore04);
  fb_gotov_K_zagruzke(StrPh:=gotov_K_zagruzke);
  fb_dPmg_Top(StrPh:=dPmg_Top);
  fb_Mv_Error(StrPh:=Mv_Error);
  fb_AutoPNS_start(StrPh:=AutoPNS_start, alg:=algoritms.autoPns);

  StrAlg.CanRun := StrAlg.inCanRun;
  StrAlg.OpcCommandsDisabled := StrAlg.inOpcCommandsDisabled;
  IF StrAlg.isRuning THEN
      (* если мв не завершен - включаем таймер *)
      IF NOT mvOn.top THEN
          runPhase(timer25);
      END_IF;

      (* если мв не заврешен - включаем таймер *)
      IF NOT mvOn.top THEN
          runPhase(timer3);
      END_IF;

      (* мв не запущен - запускаем мв *)
      IF NOT mvOn.start THEN
          runPhase(mvOn);
      END_IF;

      (* мв завершен *)
      IF mvOn.top  THEN
      (*если проверка пгнс не включена - включаем *)
          IF NOT pGNSmore04.start (*AND ((algManager.mode = modegpa.MODE_PUSKAP_R) OR (algManager.mode = modegpa.MODE_PUSKPP_R))*) THEN
              runPhase(pGNSmore04);
          END_IF;

          (*kakoito flag, hz zachem on
          IF NOT autoAVOM_canrun_flag THEN
              algoritms.S_AutoAVOM.CanRun:=TRUE;
              autoAVOM_canrun_flag:=TRUE;
          END_IF;*)
          resetPhase(timer3);
          resetPhase(timer25);
          Mv_Error.error := FALSE;
          runPhase(gotov_K_zagruzke);
          IF NOT dPmg_Top.start (*AND ((algManager.mode = modegpa.MODE_PUSKAP_R) OR (algManager.mode = modegpa.MODE_PUSKPP_R))*) THEN
              runPhase(dPmg_Top);
          END_IF;

          runDiProtection(protections.mvOff);
          runDiProtection(protections.Off_avar_vikluchatel);
          runDiProtection(protections.Reg_vozb_off);
          ELSIF NOT mvOn.top AND timer3.top THEN
  		Mv_Error.error := TRUE;
      END_IF;

      IF	dPmg_Top.start AND NOT dPmg_Top.top THEN
  	    IF	NOT IM.SingleSignals.dP_maslo_gaz_Less100.Q AND IM.SingleSignals.dP_maslo_gaz_Less100.status = 1 AND ai.dPmaslo_gaz.value > 150.0	THEN
  		    dPmg_Top.top:=TRUE;
  		    runAiProtection(protections.dPmaslo_gaz);
  		    runDiProtection(protections.dPmaslo_gaz_less100);
  		    resetAiProtection(protections.Pgaza_na_vhode_nagnetatelia_GPA_STOP);
  		    resetAiProtection(protections.Pgaza_na_vyhode_nagnetatelia_GPA_STOP);
  		    (*algoritms.autoNu_2.CanRun:=TRUE;
  		    algoritms.autoNu_2.run (); не понимаю*)
  	    END_IF;
      END_IF;

      IF	pGNSmore04.start AND NOT pGNSmore04.top THEN
  	    IF 	ai.Pmasla_posle_GNS.interval	>=statusAi.NORMAL AND ai.Pmasla_posle_GNS.value	 > 400.0 THEN
  	  	    pGNSmore04.top:=TRUE;
  	    END_IF;
      END_IF;

      IF	pGNSmore04.top AND gotov_K_zagruzke.top AND dPmg_Top.top (*AND algManager.mode = modegpa.MODE_PUSKAP_R) OR (algManager.mode = modegpa.MODE_PUSKPP_R)))*) OR
  	    gotov_K_zagruzke.top (*AND ((algManager.mode = modegpa.MODE_PUSKV_R) OR (algManager.mode = modegpa.MODE_I))))*) AND NOT AutoPNS_start.top  THEN
  	    algoritms.AutoPns.CanRun :=TRUE;
  	   (*algoritms.AutoPNS_Start.run();*)
  	    AutoPNS_start.top:=TRUE;
      END_IF;
      IF	timer25.top AND Mv_Error.error THEN
  	algoritms.ao.CanRun:=TRUE;
  	(*algoritms.ao.run ();*)
      END_IF;

      (*StrAlg.isEnded:= avom1cmdOff.top AND avom2cmdOff.top;*)
  END_IF;
  StrAlg.CanRun := StrAlg.inCanRun;
  StrAlg.OpcCommandsDisabled := StrAlg.inOpcCommandsDisabled;

  (* ---- Если управление с ВУ заблокировано, то  передаем команду из алгоритма ---- *)
  IF StrAlg.inOpcCommandsDisabled THEN
  	StrAlg.inCommand := StrAlg.inCommand_Alg;
  ELSE (* иначе передаем команду с АРМа*)
  	StrAlg.inCommand := StrAlg.inCommand_ARM;
  END_IF;

  _sunpackerCommand(command := StrAlg.inCommand);
  	source := _sunpackerCommand.source;
  	cmd := _sunpackerCommand.cmd;

  IF cmd <> 0 AND lastCmd <> cmd AND (((NOT StrAlg.opcCommandsDisabled) AND source > 0) OR source = 0) then
  	CASE BYTE_TO_INT(cmd) OF
  		(*cmdRun*) 1: 	IF (StrAlg.CanRun) THEN
  					StrAlg.isRuning := TRUE;
  					StrAlg.isEnded := FALSE;
  					StrAlg.hasError := FALSE;
  					(*****************       OnRun       *****************)
                                                    algManager.nMode:=ModeGpa.MODE_PUSK_FIRST_FAZA2;

                                                    (*runPhase(timer120);
                                                    runPhase(timer5);
                                                    runPhase(Shup);
                                                    resetAiProtection(protections.dPmaslo_gaz);
                                                    resetDiProtection(protections.dPmaslo_gaz_less100);*)

  					cmd_for_Status := cmd;
  					source_for_Status := source;
  					command_error_for_Status := 0;
  				ELSE
  					StrAlg.isRuning := FALSE;
  					StrAlg.isEnded := FALSE;
  					StrAlg.hasError := FALSE;

  					cmd_for_Status := 0;
  					source_for_Status := source;
  					command_error_for_Status := cmd;
  				END_IF;
  		(*cmdReset*) 2: 	StrAlg.isRuning := FALSE;
  				StrAlg.isEnded := FALSE;
  				StrAlg.hasError 	:= FALSE;

                                           (*****************       OnReset       *****************)
                                          waitReset(IN:=FALSE);
                                          StrAlg.inCanRun:=FALSE;

                                          (*resetPhase(timer5);
                                          resetPhase(Shup);
                                          resetPhase(timer120);
                                          resetPhase(Net_Chast);
                                          resetPhase(mvOn);
                                          resetPhase(pGNSmore04);
                                          resetPhase(gotov_K_zagruzke);
                                          resetPhase(dPmg_Top);
                                          resetPhase(AutoPNS_Start);*)

                                          StrAlg.inOpcCommandsDisabled:=FALSE;

  				cmd_for_Status := cmd;
  				source_for_Status := source;
  				command_error_for_Status := 0;
  	END_CASE;
  	resetCmdTimer(IN := false);
  	resetCmdTimerPriznak := TRUE;
  END_IF;
  lastCmd := cmd;

  resetCmdTimer(IN := resetCmdTimerPriznak, PT := T#5S);
  IF resetCmdTimer.Q THEN
  	resetCmdTimerPriznak := FALSE;
  	source_for_Status := 0;
  	cmd_for_Status := 0;
  	command_error_for_Status := 0;
  END_IF;

  StrAlg.Start:= timer25.errorStatus
              OR timer3.errorStatus
              OR mvOn.errorStatus
              OR pGNSmore04.errorStatus
              OR gotov_K_zagruzke.errorStatus
              OR dPmg_Top.errorStatus
              OR Mv_Error.errorStatus
              OR AutoPNS_Start.errorStatus;

  (*TODO: TYPE PROGRAM CODE HERE*)
  StrAlg.status :=  SHL(BYTE_TO_DWORD(source_for_Status), 29)
  			OR SHL(BYTE_TO_DWORD(cmd_for_Status), 26)
  			OR SHL(BYTE_TO_DWORD(command_error_for_Status), 23)
  			OR SHL(BOOL_TO_DWORD(StrAlg.OpcCommandsDisabled ), 21)
  			OR SHL(BOOL_TO_DWORD(StrAlg.hasError),4)
  			OR SHL(BOOL_TO_DWORD(StrAlg.CanRun),2)
  			OR SHL(BOOL_TO_DWORD(StrAlg.isEnded),1)
  			OR BOOL_TO_DWORD(StrAlg.isRuning);
END_FUNCTION_BLOCK

FUNCTION_BLOCK fb_AOSourceMlp
  VAR_IN_OUT
    OutCurrent : TDoubleData;
    strAO : struct_AO;
  END_VAR
  VAR
    _sunpackerCommand : fb_sunpackerCommand;
    source : BYTE;
    source_for_Status : BYTE;
    cmd : BYTE;
    cmd_for_Status : BYTE;
    lastCmd : BYTE;
    command_error_for_Status : BYTE;
    resetCmdTimer : TON;
    resetCmdTimerPriznak : BOOL;
    secondTack : BOOL;
    inOpcCommandsDisabled : BOOL;
  END_VAR
  VAR_INPUT RETAIN
    retainLL : LREAL;
    retainHL : LREAL;
  END_VAR

  IF NOT secondTack THEN
            IF (strAO.newLL <> retainLL) AND (retainLL <> 0.0) THEN  strAO.LL := retainLL;
            ELSE strAO.LL:= strAO.newLL; END_IF;
  	IF (strAO.newHL <> retainHL) AND (retainHL <> 0.0) THEN  strAO.HL := retainHL;
            ELSE strAO.HL:= strAO.newHL; END_IF;

  	secondTack  := FALSE;
  END_IF;
  strAO.blConnect :=(UINT_TO_WORD(OutCurrent.wFlags) AND 16#0040) <> 0;
  strAO.OpcCommandsDisabled := inOpcCommandsDisabled;

  _sunpackerCommand(command := strAO.inCommand);
  	source := _sunpackerCommand.source;
  	cmd := _sunpackerCommand.cmd;

  IF cmd <> 0 AND lastCmd <> cmd and (((NOT strAO.opcCommandsDisabled) AND source > 0) OR source = 0) then
  	CASE BYTE_TO_INT(cmd) OF
  	(*cmd_ChangeValue*) 1 : 	IF ((NOT strAO.newLL_ISVALIDREF) OR (strAO.nValue >= strAO.LL)) AND
                                             ((NOT strAO.newHL_ISVALIDREF) OR (strAO.nValue <= strAO.HL) ) THEN
  					strAO.Value := strAO.nValue;
  				END_IF;
  	(*cmd_ChangeLimits*) 2 : 	strAO.LL := strAO.newLL; retainLL:= strAO.LL;
  				strAO.HL := strAO.newHL; retainHL:= strAO.HL;
  	END_CASE;
  	source_for_Status := source;
  	cmd_for_Status := cmd;
  	command_error_for_Status := 0;
  	resetCmdTimer(IN := FALSE);
  	resetCmdTimerPriznak := TRUE;
  END_IF;
  lastCmd := cmd;

  IF (strAO.HL <> strAO.LL) THEN
  	OutCurrent.dblValue := ((strAO.Value - strAO.LL) * (strAO.outHL-strAO.outLL)/(strAO.HL - strAO.LL )) + strAO.outLL;
  END_IF;

  resetCmdTimer(IN := resetCmdTimerPriznak, PT := T#5S);
  IF resetCmdTimer.Q THEN
  	resetCmdTimerPriznak := FALSE;
  	source_for_Status := 0;
  	cmd_for_Status := 0;
  	command_error_for_Status := 0;
  END_IF;

  strAO.status := SHL(BYTE_TO_DWORD(source_for_Status), 29)
  			OR SHL(BYTE_TO_DWORD(cmd_for_Status), 26)
  			OR SHL(BYTE_TO_DWORD(command_error_for_Status), 23)
  			OR SHL(BOOL_TO_DWORD(strAO.OpcCommandsDisabled ), 21);
END_FUNCTION_BLOCK

FUNCTION_BLOCK proc_AO
  VAR
    fb_Reserv_AO_1 : fb_AOSourceMlp;
    fb_Reserv_AO_2 : fb_AOSourceMlp;
  END_VAR
  VAR_EXTERNAL
    ao : AOConfig;
    arAOUT_0 : TDoubleData;
    arAOUT_1 : TDoubleData;
  END_VAR

  (* Циклический опрос. Входные аналоговые параметры *)

  (* Модуль A10 *)

  (* [A10-1, AO0] Резерв (A10) *)
  fb_Reserv_AO_1(OutCurrent := arAOUT_0, strAO := ao.Reserv_AO_1);

  (* [A10-1, AO1] Резерв (A10) *)
  fb_Reserv_AO_2(OutCurrent := arAOUT_1, strAO := ao.Reserv_AO_2);
END_FUNCTION_BLOCK

FUNCTION EnableAiLimits : BOOL
  VAR_IN_OUT
    ai : AiConfig;
  END_VAR

  ai.Pmasla_posle_GNS.Disabled_LA:=FALSE;
   ai.Pmasla_posle_GNS.Disabled_LW:=FALSE;
   ai.Pmasla_posle_NU.Disabled_LW:=FALSE;
   ai.Tmasla_MB.Disabled_LA:=FALSE;
   ai.Tmasla_MB.Disabled_LW:=FALSE;
END_FUNCTION

FUNCTION DisableAiLimits : BOOL
  VAR_IN_OUT
    ai : AiConfig;
  END_VAR

  ai.Pmasla_posle_GNS.Disabled_LA:=TRUE;
  ai.Pmasla_posle_GNS.Disabled_LW:=TRUE;
  ai.Pmasla_posle_NU.Disabled_LW:=TRUE;
  ai.Tmasla_MB.Disabled_LA:=TRUE;
  ai.Tmasla_MB.Disabled_LW:=TRUE;
END_FUNCTION

FUNCTION_BLOCK TestProtectionAlg
  VAR_IN_OUT
    StrAlg : struct_Alg;
  END_VAR
  VAR
    _sunpackerCommand : fb_sunpackerCommand;
    source : BYTE;
    cmd : BYTE;
    lastCmd : BYTE;
    source_for_Status : BYTE;
    cmd_for_Status : BYTE;
    command_error_for_Status : BYTE;
    resetCmdTimer : TON;
    resetCmdTimerPriznak : BOOL;
  END_VAR
  VAR_EXTERNAL
    ai : AiConfig;
    protectManager : struct_ProtectionsManager;
    algManager : struct_AlgoritmsManager;
    ModeGpa : TYPE_ModeGpa;
    PMcommand : TYPE_CommandsPotectionsManager;
    IM : ImConfig;
  END_VAR

  StrAlg.CanRun := StrAlg.inCanRun;
  StrAlg.OpcCommandsDisabled := StrAlg.inOpcCommandsDisabled;

  (* ---- Если управление с ВУ заблокировано, то передаем команду из алгоритма ---- *)
  IF StrAlg.inOpcCommandsDisabled THEN
  	StrAlg.inCommand := StrAlg.inCommand_Alg;
  ELSE (* иначе передаем команду с АРМа*)
  	StrAlg.inCommand := StrAlg.inCommand_ARM;
  END_IF;

  _sunpackerCommand(command := StrAlg.inCommand);
  	source := _sunpackerCommand.source;
  	cmd := _sunpackerCommand.cmd;

  IF cmd <> 0 AND lastCmd <> cmd AND (((NOT StrAlg.opcCommandsDisabled) AND source > 0) OR source = 0) then
  	CASE BYTE_TO_INT(cmd) OF
  		(*cmdRun*) 1: 	IF (StrAlg.CanRun) THEN
  					StrAlg.isRuning := TRUE;
  					StrAlg.isEnded := FALSE;
  					StrAlg.hasError 	:= FALSE;
                                               (*****************       OnRun       *****************)
                                                        algManager.nMode:=ModeGpa.MODE_TESTAZ;
                                                        protectManager.inCommand:=PMcommand.CheckProtections;
  					    EnableAiLimits(ai);
                                                        (*IM.SingleSignals.P_oil_low.Disabled_Sig:=FALSE;*)
                                                        (*IM.SingleSignals.dP_oilgaz_low.Disabled_Sig:=FALSE;*)
                                                    (*StrAlg.inOpcCommandsDisabled:=FALSE;*)
  					cmd_for_Status := cmd;
  					source_for_Status := source;
  					command_error_for_Status := 0;
  				ELSE
  					StrAlg.isRuning := FALSE;
  					StrAlg.isEnded := FALSE;
  					StrAlg.hasError 	:= FALSE;

  					cmd_for_Status := 0;
  					source_for_Status := source;
  					command_error_for_Status := cmd;
  				END_IF;
  		(*cmdReset*) 2: 	StrAlg.isRuning := FALSE;
  				StrAlg.isEnded := FALSE;
  				StrAlg.hasError 	:= FALSE;
                                          (*****************       OnReset       *****************)
                                                    DisableAiLimits(ai);
                                                    (*IM.SingleSignals.P_oil_low.Disabled_Sig:=TRUE;
                                                    IM.SingleSignals.dP_oilgaz_low.Disabled_Sig:=TRUE;*)
                                                    protectManager.inCommand:=PMcommand.RestartAllProtections;
                                                    algManager.nMode:=ModeGpa.MODE_STOP;

  				cmd_for_Status := cmd;
  				source_for_Status := source;
  				command_error_for_Status := 0;
  	END_CASE;
  	resetCmdTimer(IN := false);
  	resetCmdTimerPriznak := TRUE;
  END_IF;
  lastCmd := cmd;

  resetCmdTimer(IN := resetCmdTimerPriznak, PT := T#5S);
  IF resetCmdTimer.Q THEN
  	resetCmdTimerPriznak := FALSE;
  	source_for_Status := 0;
  	cmd_for_Status := 0;
  	command_error_for_Status := 0;
  END_IF;
